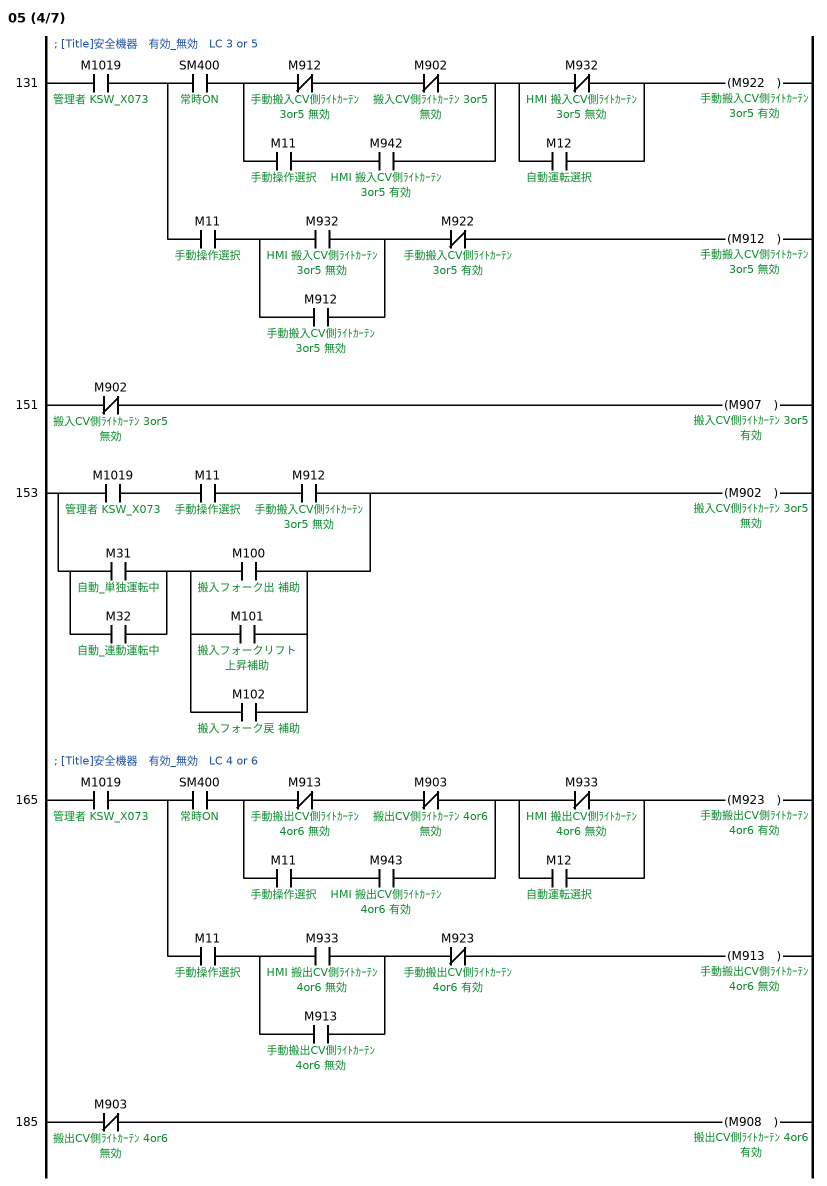
; [Title]安全機器　有効_無効　LC 3 or 5
131   LD      M1019  ; 管理者 KSW_X073
      MPS
      AND     SM400  ; 常時ON
      LDI     M912  ; 手動搬入CV側ﾗｲﾄｶｰﾃﾝ 3or5 無効
      ANI     M902  ; 搬入CV側ﾗｲﾄｶｰﾃﾝ 3or5 無効
      LD      M11  ; 手動操作選択
      AND     M942  ; HMI 搬入CV側ﾗｲﾄｶｰﾃﾝ 3or5 有効
      ORB
      ANB
      LDI     M932  ; HMI 搬入CV側ﾗｲﾄｶｰﾃﾝ 3or5 無効
      OR      M12  ; 自動運転選択
      ANB
      OUT     M922  ; 手動搬入CV側ﾗｲﾄｶｰﾃﾝ 3or5 有効
      MPP
      AND     M11  ; 手動操作選択
      LD      M932  ; HMI 搬入CV側ﾗｲﾄｶｰﾃﾝ 3or5 無効
      OR      M912  ; 手動搬入CV側ﾗｲﾄｶｰﾃﾝ 3or5 無効
      ANB
      ANI     M922  ; 手動搬入CV側ﾗｲﾄｶｰﾃﾝ 3or5 有効
      OUT     M912  ; 手動搬入CV側ﾗｲﾄｶｰﾃﾝ 3or5 無効
151   LDI     M902  ; 搬入CV側ﾗｲﾄｶｰﾃﾝ 3or5 無効
      OUT     M907  ; 搬入CV側ﾗｲﾄｶｰﾃﾝ 3or5 有効
153   LD      M1019  ; 管理者 KSW_X073
      AND     M11  ; 手動操作選択
      AND     M912  ; 手動搬入CV側ﾗｲﾄｶｰﾃﾝ 3or5 無効
      LD      M31  ; 自動_単独運転中
      OR      M32  ; 自動_連動運転中
      LD      M100  ; 搬入フォーク出 補助
      OR      M101  ; 搬入フォークリフト 上昇補助
      OR      M102  ; 搬入フォーク戻 補助
      ANB
      ORB
      OUT     M902  ; 搬入CV側ﾗｲﾄｶｰﾃﾝ 3or5 無効
; [Title]安全機器　有効_無効　LC 4 or 6
165   LD      M1019  ; 管理者 KSW_X073
      MPS
      AND     SM400  ; 常時ON
      LDI     M913  ; 手動搬出CV側ﾗｲﾄｶｰﾃﾝ 4or6 無効
      ANI     M903  ; 搬出CV側ﾗｲﾄｶｰﾃﾝ 4or6 無効
      LD      M11  ; 手動操作選択
      AND     M943  ; HMI 搬出CV側ﾗｲﾄｶｰﾃﾝ 4or6 有効
      ORB
      ANB
      LDI     M933  ; HMI 搬出CV側ﾗｲﾄｶｰﾃﾝ 4or6 無効
      OR      M12  ; 自動運転選択
      ANB
      OUT     M923  ; 手動搬出CV側ﾗｲﾄｶｰﾃﾝ 4or6 有効
      MPP
      AND     M11  ; 手動操作選択
      LD      M933  ; HMI 搬出CV側ﾗｲﾄｶｰﾃﾝ 4or6 無効
      OR      M913  ; 手動搬出CV側ﾗｲﾄｶｰﾃﾝ 4or6 無効
      ANB
      ANI     M923  ; 手動搬出CV側ﾗｲﾄｶｰﾃﾝ 4or6 有効
      OUT     M913  ; 手動搬出CV側ﾗｲﾄｶｰﾃﾝ 4or6 無効
185   LDI     M903  ; 搬出CV側ﾗｲﾄｶｰﾃﾝ 4or6 無効
      OUT     M908  ; 搬出CV側ﾗｲﾄｶｰﾃﾝ 4or6 有効
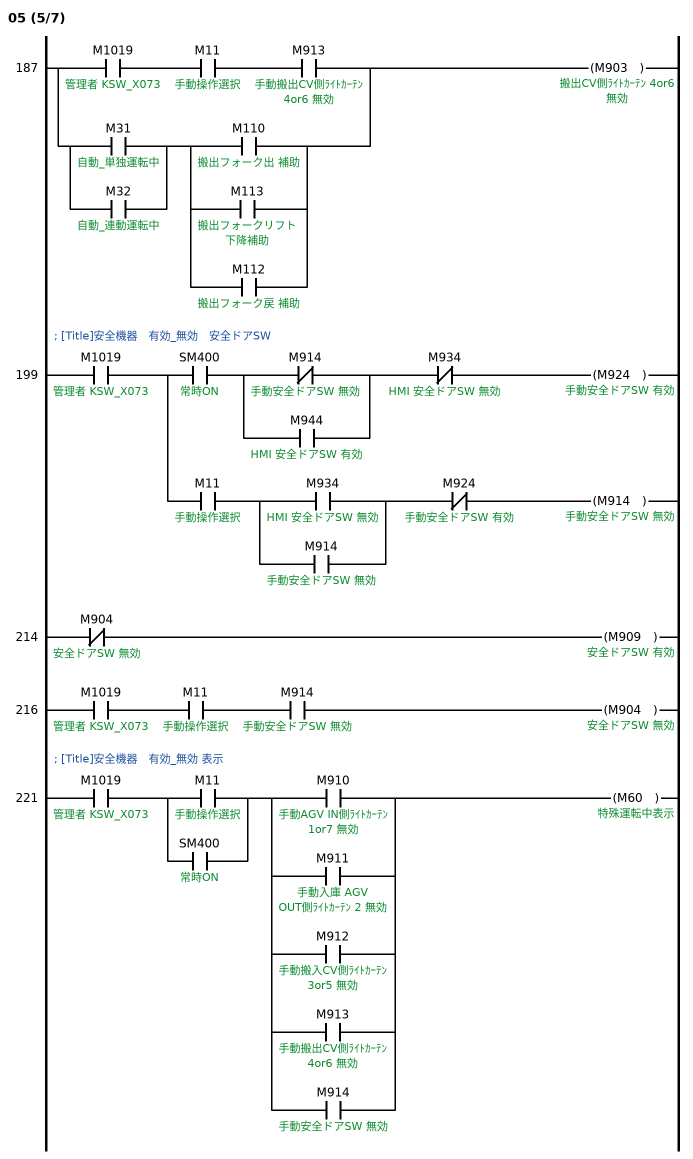
187   LD      M1019  ; 管理者 KSW_X073
      AND     M11  ; 手動操作選択
      AND     M913  ; 手動搬出CV側ﾗｲﾄｶｰﾃﾝ 4or6 無効
      LD      M31  ; 自動_単独運転中
      OR      M32  ; 自動_連動運転中
      LD      M110  ; 搬出フォーク出 補助
      OR      M113  ; 搬出フォークリフト 下降補助
      OR      M112  ; 搬出フォーク戻 補助
      ANB
      ORB
      OUT     M903  ; 搬出CV側ﾗｲﾄｶｰﾃﾝ 4or6 無効
; [Title]安全機器　有効_無効　安全ドアSW
199   LD      M1019  ; 管理者 KSW_X073
      MPS
      AND     SM400  ; 常時ON
      LDI     M914  ; 手動安全ドアSW 無効
      OR      M944  ; HMI 安全ドアSW 有効
      ANB
      ANI     M934  ; HMI 安全ドアSW 無効
      OUT     M924  ; 手動安全ドアSW 有効
      MPP
      AND     M11  ; 手動操作選択
      LD      M934  ; HMI 安全ドアSW 無効
      OR      M914  ; 手動安全ドアSW 無効
      ANB
      ANI     M924  ; 手動安全ドアSW 有効
      OUT     M914  ; 手動安全ドアSW 無効
214   LDI     M904  ; 安全ドアSW 無効
      OUT     M909  ; 安全ドアSW 有効
216   LD      M1019  ; 管理者 KSW_X073
      AND     M11  ; 手動操作選択
      AND     M914  ; 手動安全ドアSW 無効
      OUT     M904  ; 安全ドアSW 無効
; [Title]安全機器　有効_無効 表示
221   LD      M1019  ; 管理者 KSW_X073
      LD      M11  ; 手動操作選択
      OR      SM400  ; 常時ON
      ANB
      LD      M910  ; 手動AGV IN側ﾗｲﾄｶｰﾃﾝ 1or7 無効
      OR      M911  ; 手動入庫 AGV OUT側ﾗｲﾄｶｰﾃﾝ 2 無効
      OR      M912  ; 手動搬入CV側ﾗｲﾄｶｰﾃﾝ 3or5 無効
      OR      M913  ; 手動搬出CV側ﾗｲﾄｶｰﾃﾝ 4or6 無効
      OR      M914  ; 手動安全ドアSW 無効
      ANB
      OUT     M60  ; 特殊運転中表示
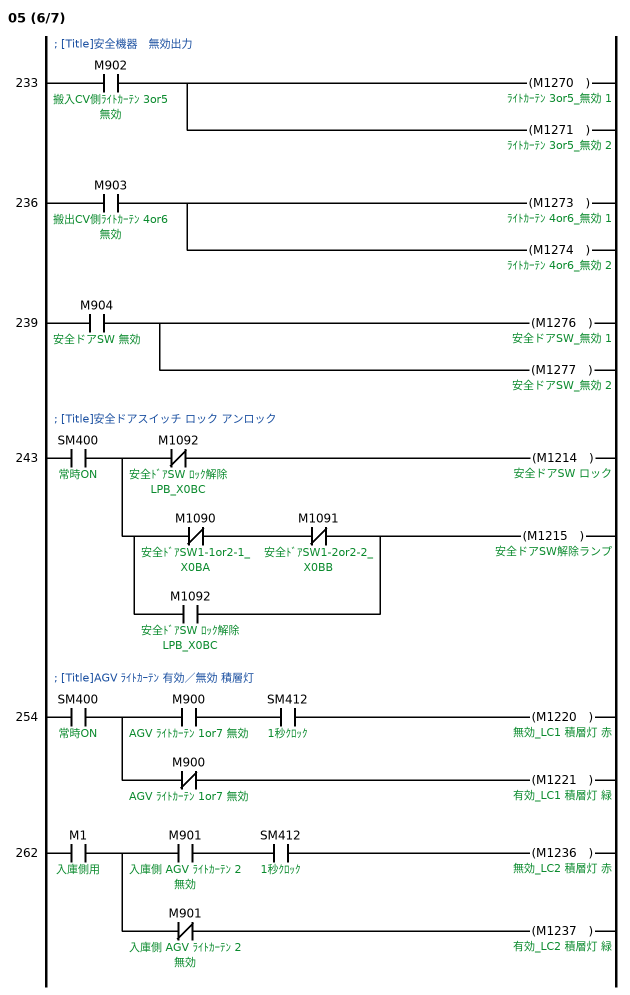
; [Title]安全機器　無効出力
233   LD      M902  ; 搬入CV側ﾗｲﾄｶｰﾃﾝ 3or5 無効
      OUT     M1270  ; ﾗｲﾄｶｰﾃﾝ 3or5_無効 1
      OUT     M1271  ; ﾗｲﾄｶｰﾃﾝ 3or5_無効 2
236   LD      M903  ; 搬出CV側ﾗｲﾄｶｰﾃﾝ 4or6 無効
      OUT     M1273  ; ﾗｲﾄｶｰﾃﾝ 4or6_無効 1
      OUT     M1274  ; ﾗｲﾄｶｰﾃﾝ 4or6_無効 2
239   LD      M904  ; 安全ドアSW 無効
      OUT     M1276  ; 安全ドアSW_無効 1
      OUT     M1277  ; 安全ドアSW_無効 2
; [Title]安全ドアスイッチ ロック アンロック
243   LD      SM400  ; 常時ON
      MPS
      ANI     M1092  ; 安全ﾄﾞｱSW ﾛｯｸ解除 LPB_X0BC
      OUT     M1214  ; 安全ドアSW ロック
      MPP
      LDI     M1090  ; 安全ﾄﾞｱSW1-1or2-1_X0BA
      ANI     M1091  ; 安全ﾄﾞｱSW1-2or2-2_X0BB
      OR      M1092  ; 安全ﾄﾞｱSW ﾛｯｸ解除 LPB_X0BC
      ANB
      OUT     M1215  ; 安全ドアSW解除ランプ
; [Title]AGV ﾗｲﾄｶｰﾃﾝ 有効／無効 積層灯
254   LD      SM400  ; 常時ON
      MPS
      AND     M900  ; AGV ﾗｲﾄｶｰﾃﾝ 1or7 無効
      AND     SM412  ; 1秒ｸﾛｯｸ
      OUT     M1220  ; 無効_LC1 積層灯 赤
      MPP
      ANI     M900  ; AGV ﾗｲﾄｶｰﾃﾝ 1or7 無効
      OUT     M1221  ; 有効_LC1 積層灯 緑
262   LD      M1  ; 入庫側用
      MPS
      AND     M901  ; 入庫側 AGV ﾗｲﾄｶｰﾃﾝ 2 無効
      AND     SM412  ; 1秒ｸﾛｯｸ
      OUT     M1236  ; 無効_LC2 積層灯 赤
      MPP
      ANI     M901  ; 入庫側 AGV ﾗｲﾄｶｰﾃﾝ 2 無効
      OUT     M1237  ; 有効_LC2 積層灯 緑
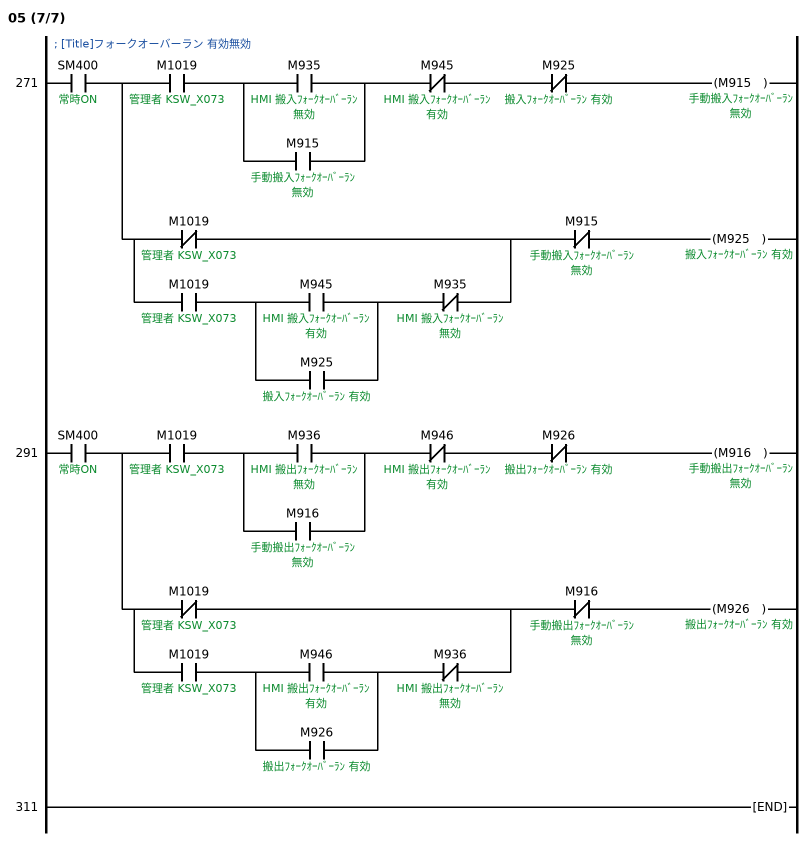
; [Title]フォークオーバーラン 有効無効
271   LD      SM400  ; 常時ON
      MPS
      AND     M1019  ; 管理者 KSW_X073
      LD      M935  ; HMI 搬入ﾌｫｰｸｵｰﾊﾞｰﾗﾝ 無効
      OR      M915  ; 手動搬入ﾌｫｰｸｵｰﾊﾞｰﾗﾝ 無効
      ANB
      ANI     M945  ; HMI 搬入ﾌｫｰｸｵｰﾊﾞｰﾗﾝ 有効
      ANI     M925  ; 搬入ﾌｫｰｸｵｰﾊﾞｰﾗﾝ 有効
      OUT     M915  ; 手動搬入ﾌｫｰｸｵｰﾊﾞｰﾗﾝ 無効
      MPP
      LDI     M1019  ; 管理者 KSW_X073
      LD      M1019  ; 管理者 KSW_X073
      LD      M945  ; HMI 搬入ﾌｫｰｸｵｰﾊﾞｰﾗﾝ 有効
      OR      M925  ; 搬入ﾌｫｰｸｵｰﾊﾞｰﾗﾝ 有効
      ANB
      ANI     M935  ; HMI 搬入ﾌｫｰｸｵｰﾊﾞｰﾗﾝ 無効
      ORB
      ANB
      ANI     M915  ; 手動搬入ﾌｫｰｸｵｰﾊﾞｰﾗﾝ 無効
      OUT     M925  ; 搬入ﾌｫｰｸｵｰﾊﾞｰﾗﾝ 有効
291   LD      SM400  ; 常時ON
      MPS
      AND     M1019  ; 管理者 KSW_X073
      LD      M936  ; HMI 搬出ﾌｫｰｸｵｰﾊﾞｰﾗﾝ 無効
      OR      M916  ; 手動搬出ﾌｫｰｸｵｰﾊﾞｰﾗﾝ 無効
      ANB
      ANI     M946  ; HMI 搬出ﾌｫｰｸｵｰﾊﾞｰﾗﾝ 有効
      ANI     M926  ; 搬出ﾌｫｰｸｵｰﾊﾞｰﾗﾝ 有効
      OUT     M916  ; 手動搬出ﾌｫｰｸｵｰﾊﾞｰﾗﾝ 無効
      MPP
      LDI     M1019  ; 管理者 KSW_X073
      LD      M1019  ; 管理者 KSW_X073
      LD      M946  ; HMI 搬出ﾌｫｰｸｵｰﾊﾞｰﾗﾝ 有効
      OR      M926  ; 搬出ﾌｫｰｸｵｰﾊﾞｰﾗﾝ 有効
      ANB
      ANI     M936  ; HMI 搬出ﾌｫｰｸｵｰﾊﾞｰﾗﾝ 無効
      ORB
      ANB
      ANI     M916  ; 手動搬出ﾌｫｰｸｵｰﾊﾞｰﾗﾝ 無効
      OUT     M926  ; 搬出ﾌｫｰｸｵｰﾊﾞｰﾗﾝ 有効
311   END
END_PROGRAM

PROGRAM 09  // Alram
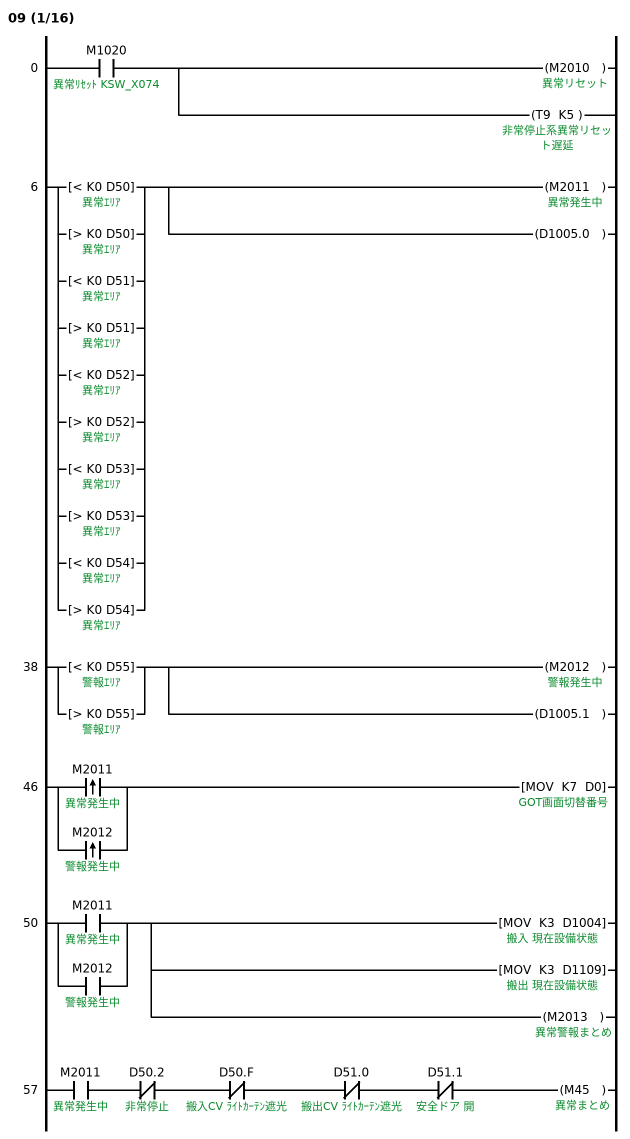
0     LD      M1020  ; 異常ﾘｾｯﾄ KSW_X074
      OUT     M2010  ; 異常リセット
      OUT     T9 K5  ; 非常停止系異常リセット遅延
6     LD<     K0 D50  ; 異常ｴﾘｱ
      OR>     K0 D50  ; 異常ｴﾘｱ
      OR<     K0 D51  ; 異常ｴﾘｱ
      OR>     K0 D51  ; 異常ｴﾘｱ
      OR<     K0 D52  ; 異常ｴﾘｱ
      OR>     K0 D52  ; 異常ｴﾘｱ
      OR<     K0 D53  ; 異常ｴﾘｱ
      OR>     K0 D53  ; 異常ｴﾘｱ
      OR<     K0 D54  ; 異常ｴﾘｱ
      OR>     K0 D54  ; 異常ｴﾘｱ
      OUT     M2011  ; 異常発生中
      OUT     D1005.0
38    LD<     K0 D55  ; 警報ｴﾘｱ
      OR>     K0 D55  ; 警報ｴﾘｱ
      OUT     M2012  ; 警報発生中
      OUT     D1005.1
46    LDP     M2011  ; 異常発生中
      ORP     M2012  ; 警報発生中
      MOV     K7 D0  ; GOT画面切替番号
50    LD      M2011  ; 異常発生中
      OR      M2012  ; 警報発生中
      MOV     K3 D1004  ; 搬入 現在設備状態
      MOV     K3 D1109  ; 搬出 現在設備状態
      OUT     M2013  ; 異常警報まとめ
57    LD      M2011  ; 異常発生中
      ANI     D50.2  ; 非常停止
      ANI     D50.F  ; 搬入CV ﾗｲﾄｶｰﾃﾝ遮光
      ANI     D51.0  ; 搬出CV ﾗｲﾄｶｰﾃﾝ遮光
      ANI     D51.1  ; 安全ドア 開
      OUT     M45  ; 異常まとめ
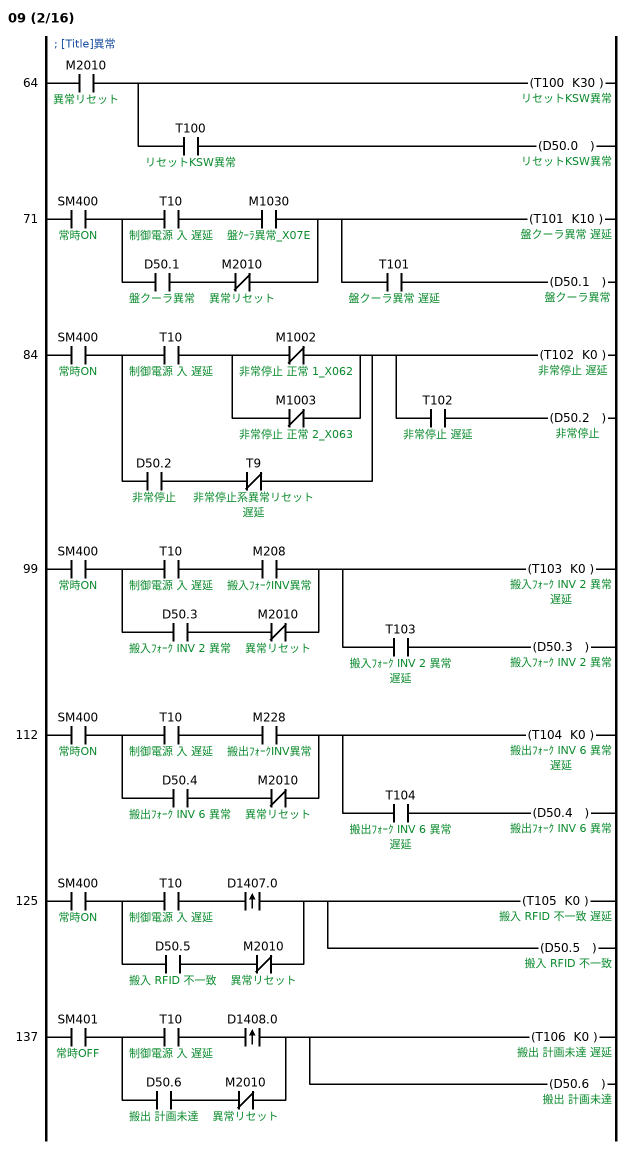
; [Title]異常
64    LD      M2010  ; 異常リセット
      OUT     T100 K30  ; リセットKSW異常
      AND     T100  ; リセットKSW異常
      OUT     D50.0  ; リセットKSW異常
71    LD      SM400  ; 常時ON
      LD      T10  ; 制御電源 入 遅延
      AND     M1030  ; 盤ｸｰﾗ異常_X07E
      LD      D50.1  ; 盤クーラ異常
      ANI     M2010  ; 異常リセット
      ORB
      ANB
      OUT     T101 K10  ; 盤クーラ異常 遅延
      AND     T101  ; 盤クーラ異常 遅延
      OUT     D50.1  ; 盤クーラ異常
84    LD      SM400  ; 常時ON
      LD      T10  ; 制御電源 入 遅延
      LDI     M1002  ; 非常停止 正常 1_X062
      ORI     M1003  ; 非常停止 正常 2_X063
      ANB
      LD      D50.2  ; 非常停止
      ANI     T9  ; 非常停止系異常リセット遅延
      ORB
      ANB
      OUT     T102 K0  ; 非常停止 遅延
      AND     T102  ; 非常停止 遅延
      OUT     D50.2  ; 非常停止
99    LD      SM400  ; 常時ON
      LD      T10  ; 制御電源 入 遅延
      AND     M208  ; 搬入ﾌｫｰｸINV異常
      LD      D50.3  ; 搬入ﾌｫｰｸ INV 2 異常
      ANI     M2010  ; 異常リセット
      ORB
      ANB
      OUT     T103 K0  ; 搬入ﾌｫｰｸ INV 2 異常 遅延
      AND     T103  ; 搬入ﾌｫｰｸ INV 2 異常 遅延
      OUT     D50.3  ; 搬入ﾌｫｰｸ INV 2 異常
112   LD      SM400  ; 常時ON
      LD      T10  ; 制御電源 入 遅延
      AND     M228  ; 搬出ﾌｫｰｸINV異常
      LD      D50.4  ; 搬出ﾌｫｰｸ INV 6 異常
      ANI     M2010  ; 異常リセット
      ORB
      ANB
      OUT     T104 K0  ; 搬出ﾌｫｰｸ INV 6 異常 遅延
      AND     T104  ; 搬出ﾌｫｰｸ INV 6 異常 遅延
      OUT     D50.4  ; 搬出ﾌｫｰｸ INV 6 異常
125   LD      SM400  ; 常時ON
      LD      T10  ; 制御電源 入 遅延
      ANDP    D1407.0
      LD      D50.5  ; 搬入 RFID 不一致
      ANI     M2010  ; 異常リセット
      ORB
      ANB
      OUT     T105 K0  ; 搬入 RFID 不一致 遅延
      OUT     D50.5  ; 搬入 RFID 不一致
137   LD      SM401  ; 常時OFF
      LD      T10  ; 制御電源 入 遅延
      ANDP    D1408.0
      LD      D50.6  ; 搬出 計画未達
      ANI     M2010  ; 異常リセット
      ORB
      ANB
      OUT     T106 K0  ; 搬出 計画未達 遅延
      OUT     D50.6  ; 搬出 計画未達
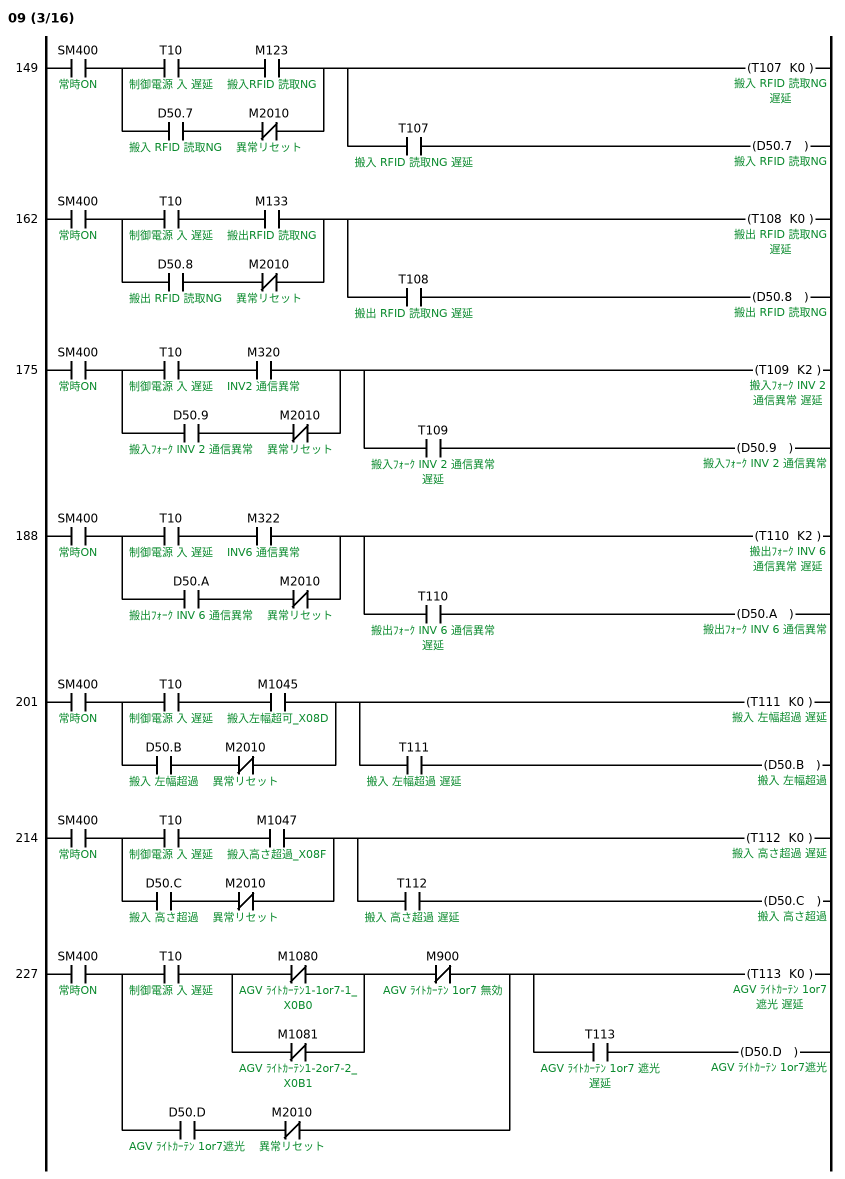
149   LD      SM400  ; 常時ON
      LD      T10  ; 制御電源 入 遅延
      AND     M123  ; 搬入RFID 読取NG
      LD      D50.7  ; 搬入 RFID 読取NG
      ANI     M2010  ; 異常リセット
      ORB
      ANB
      OUT     T107 K0  ; 搬入 RFID 読取NG 遅延
      AND     T107  ; 搬入 RFID 読取NG 遅延
      OUT     D50.7  ; 搬入 RFID 読取NG
162   LD      SM400  ; 常時ON
      LD      T10  ; 制御電源 入 遅延
      AND     M133  ; 搬出RFID 読取NG
      LD      D50.8  ; 搬出 RFID 読取NG
      ANI     M2010  ; 異常リセット
      ORB
      ANB
      OUT     T108 K0  ; 搬出 RFID 読取NG 遅延
      AND     T108  ; 搬出 RFID 読取NG 遅延
      OUT     D50.8  ; 搬出 RFID 読取NG
175   LD      SM400  ; 常時ON
      LD      T10  ; 制御電源 入 遅延
      AND     M320  ; INV2 通信異常
      LD      D50.9  ; 搬入ﾌｫｰｸ INV 2 通信異常
      ANI     M2010  ; 異常リセット
      ORB
      ANB
      OUT     T109 K2  ; 搬入ﾌｫｰｸ INV 2 通信異常 遅延
      AND     T109  ; 搬入ﾌｫｰｸ INV 2 通信異常 遅延
      OUT     D50.9  ; 搬入ﾌｫｰｸ INV 2 通信異常
188   LD      SM400  ; 常時ON
      LD      T10  ; 制御電源 入 遅延
      AND     M322  ; INV6 通信異常
      LD      D50.A  ; 搬出ﾌｫｰｸ INV 6 通信異常
      ANI     M2010  ; 異常リセット
      ORB
      ANB
      OUT     T110 K2  ; 搬出ﾌｫｰｸ INV 6 通信異常 遅延
      AND     T110  ; 搬出ﾌｫｰｸ INV 6 通信異常 遅延
      OUT     D50.A  ; 搬出ﾌｫｰｸ INV 6 通信異常
201   LD      SM400  ; 常時ON
      LD      T10  ; 制御電源 入 遅延
      AND     M1045  ; 搬入左幅超可_X08D
      LD      D50.B  ; 搬入 左幅超過
      ANI     M2010  ; 異常リセット
      ORB
      ANB
      OUT     T111 K0  ; 搬入 左幅超過 遅延
      AND     T111  ; 搬入 左幅超過 遅延
      OUT     D50.B  ; 搬入 左幅超過
214   LD      SM400  ; 常時ON
      LD      T10  ; 制御電源 入 遅延
      AND     M1047  ; 搬入高さ超過_X08F
      LD      D50.C  ; 搬入 高さ超過
      ANI     M2010  ; 異常リセット
      ORB
      ANB
      OUT     T112 K0  ; 搬入 高さ超過 遅延
      AND     T112  ; 搬入 高さ超過 遅延
      OUT     D50.C  ; 搬入 高さ超過
227   LD      SM400  ; 常時ON
      LD      T10  ; 制御電源 入 遅延
      LDI     M1080  ; AGV ﾗｲﾄｶｰﾃﾝ1-1or7-1_X0B0
      ORI     M1081  ; AGV ﾗｲﾄｶｰﾃﾝ1-2or7-2_X0B1
      ANB
      ANI     M900  ; AGV ﾗｲﾄｶｰﾃﾝ 1or7 無効
      LD      D50.D  ; AGV ﾗｲﾄｶｰﾃﾝ 1or7遮光
      ANI     M2010  ; 異常リセット
      ORB
      ANB
      OUT     T113 K0  ; AGV ﾗｲﾄｶｰﾃﾝ 1or7 遮光 遅延
      AND     T113  ; AGV ﾗｲﾄｶｰﾃﾝ 1or7 遮光 遅延
      OUT     D50.D  ; AGV ﾗｲﾄｶｰﾃﾝ 1or7遮光
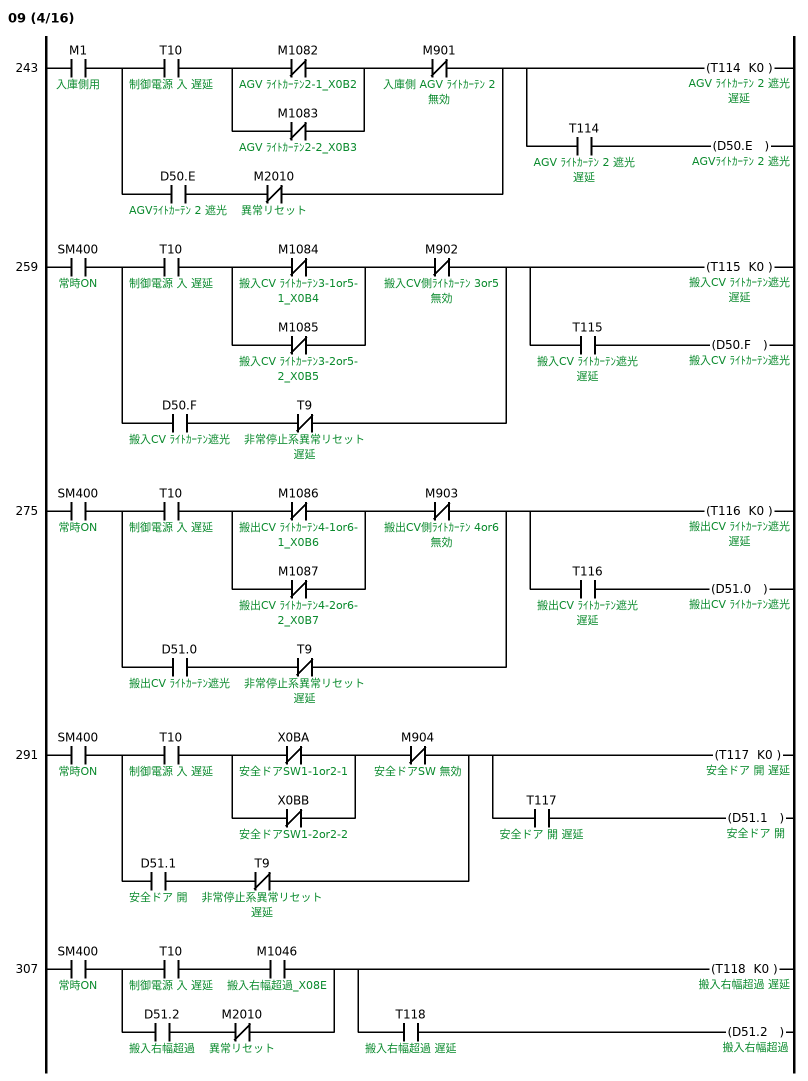
243   LD      M1  ; 入庫側用
      LD      T10  ; 制御電源 入 遅延
      LDI     M1082  ; AGV ﾗｲﾄｶｰﾃﾝ2-1_X0B2
      ORI     M1083  ; AGV ﾗｲﾄｶｰﾃﾝ2-2_X0B3
      ANB
      ANI     M901  ; 入庫側 AGV ﾗｲﾄｶｰﾃﾝ 2 無効
      LD      D50.E  ; AGVﾗｲﾄｶｰﾃﾝ 2 遮光
      ANI     M2010  ; 異常リセット
      ORB
      ANB
      OUT     T114 K0  ; AGV ﾗｲﾄｶｰﾃﾝ 2 遮光 遅延
      AND     T114  ; AGV ﾗｲﾄｶｰﾃﾝ 2 遮光 遅延
      OUT     D50.E  ; AGVﾗｲﾄｶｰﾃﾝ 2 遮光
259   LD      SM400  ; 常時ON
      LD      T10  ; 制御電源 入 遅延
      LDI     M1084  ; 搬入CV ﾗｲﾄｶｰﾃﾝ3-1or5-1_X0B4
      ORI     M1085  ; 搬入CV ﾗｲﾄｶｰﾃﾝ3-2or5-2_X0B5
      ANB
      ANI     M902  ; 搬入CV側ﾗｲﾄｶｰﾃﾝ 3or5 無効
      LD      D50.F  ; 搬入CV ﾗｲﾄｶｰﾃﾝ遮光
      ANI     T9  ; 非常停止系異常リセット遅延
      ORB
      ANB
      OUT     T115 K0  ; 搬入CV ﾗｲﾄｶｰﾃﾝ遮光 遅延
      AND     T115  ; 搬入CV ﾗｲﾄｶｰﾃﾝ遮光 遅延
      OUT     D50.F  ; 搬入CV ﾗｲﾄｶｰﾃﾝ遮光
275   LD      SM400  ; 常時ON
      LD      T10  ; 制御電源 入 遅延
      LDI     M1086  ; 搬出CV ﾗｲﾄｶｰﾃﾝ4-1or6-1_X0B6
      ORI     M1087  ; 搬出CV ﾗｲﾄｶｰﾃﾝ4-2or6-2_X0B7
      ANB
      ANI     M903  ; 搬出CV側ﾗｲﾄｶｰﾃﾝ 4or6 無効
      LD      D51.0  ; 搬出CV ﾗｲﾄｶｰﾃﾝ遮光
      ANI     T9  ; 非常停止系異常リセット遅延
      ORB
      ANB
      OUT     T116 K0  ; 搬出CV ﾗｲﾄｶｰﾃﾝ遮光 遅延
      AND     T116  ; 搬出CV ﾗｲﾄｶｰﾃﾝ遮光 遅延
      OUT     D51.0  ; 搬出CV ﾗｲﾄｶｰﾃﾝ遮光
291   LD      SM400  ; 常時ON
      LD      T10  ; 制御電源 入 遅延
      LDI     X0BA  ; 安全ドアSW1-1or2-1
      ORI     X0BB  ; 安全ドアSW1-2or2-2
      ANB
      ANI     M904  ; 安全ドアSW 無効
      LD      D51.1  ; 安全ドア 開
      ANI     T9  ; 非常停止系異常リセット遅延
      ORB
      ANB
      OUT     T117 K0  ; 安全ドア 開 遅延
      AND     T117  ; 安全ドア 開 遅延
      OUT     D51.1  ; 安全ドア 開
307   LD      SM400  ; 常時ON
      LD      T10  ; 制御電源 入 遅延
      AND     M1046  ; 搬入右幅超過_X08E
      LD      D51.2  ; 搬入右幅超過
      ANI     M2010  ; 異常リセット
      ORB
      ANB
      OUT     T118 K0  ; 搬入右幅超過 遅延
      AND     T118  ; 搬入右幅超過 遅延
      OUT     D51.2  ; 搬入右幅超過
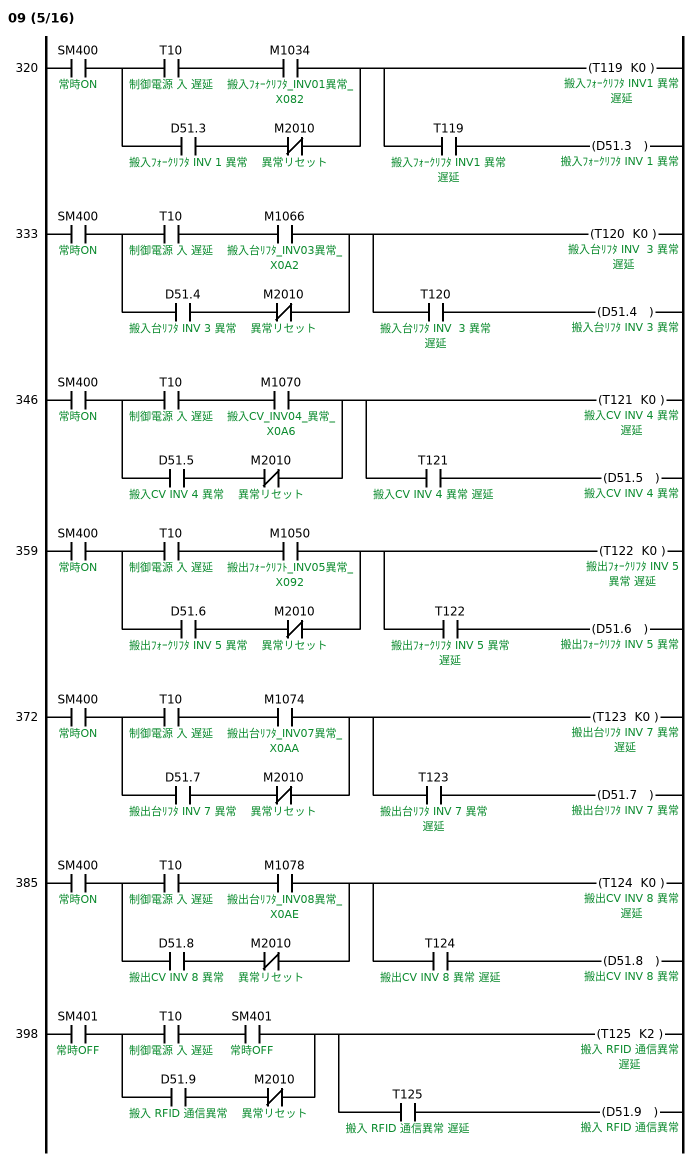
320   LD      SM400  ; 常時ON
      LD      T10  ; 制御電源 入 遅延
      AND     M1034  ; 搬入ﾌｫｰｸﾘﾌﾀ_INV01異常_X082
      LD      D51.3  ; 搬入ﾌｫｰｸﾘﾌﾀ INV 1 異常
      ANI     M2010  ; 異常リセット
      ORB
      ANB
      OUT     T119 K0  ; 搬入ﾌｫｰｸﾘﾌﾀ INV1 異常 遅延
      AND     T119  ; 搬入ﾌｫｰｸﾘﾌﾀ INV1 異常 遅延
      OUT     D51.3  ; 搬入ﾌｫｰｸﾘﾌﾀ INV 1 異常
333   LD      SM400  ; 常時ON
      LD      T10  ; 制御電源 入 遅延
      AND     M1066  ; 搬入台ﾘﾌﾀ_INV03異常_X0A2
      LD      D51.4  ; 搬入台ﾘﾌﾀ INV 3 異常
      ANI     M2010  ; 異常リセット
      ORB
      ANB
      OUT     T120 K0  ; 搬入台ﾘﾌﾀ INV  3 異常 遅延
      AND     T120  ; 搬入台ﾘﾌﾀ INV  3 異常 遅延
      OUT     D51.4  ; 搬入台ﾘﾌﾀ INV 3 異常
346   LD      SM400  ; 常時ON
      LD      T10  ; 制御電源 入 遅延
      AND     M1070  ; 搬入CV_INV04_異常_X0A6
      LD      D51.5  ; 搬入CV INV 4 異常
      ANI     M2010  ; 異常リセット
      ORB
      ANB
      OUT     T121 K0  ; 搬入CV INV 4 異常 遅延
      AND     T121  ; 搬入CV INV 4 異常 遅延
      OUT     D51.5  ; 搬入CV INV 4 異常
359   LD      SM400  ; 常時ON
      LD      T10  ; 制御電源 入 遅延
      AND     M1050  ; 搬出ﾌｫｰｸﾘﾌﾄ_INV05異常_X092
      LD      D51.6  ; 搬出ﾌｫｰｸﾘﾌﾀ INV 5 異常
      ANI     M2010  ; 異常リセット
      ORB
      ANB
      OUT     T122 K0  ; 搬出ﾌｫｰｸﾘﾌﾀ INV 5 異常 遅延
      AND     T122  ; 搬出ﾌｫｰｸﾘﾌﾀ INV 5 異常 遅延
      OUT     D51.6  ; 搬出ﾌｫｰｸﾘﾌﾀ INV 5 異常
372   LD      SM400  ; 常時ON
      LD      T10  ; 制御電源 入 遅延
      AND     M1074  ; 搬出台ﾘﾌﾀ_INV07異常_X0AA
      LD      D51.7  ; 搬出台ﾘﾌﾀ INV 7 異常
      ANI     M2010  ; 異常リセット
      ORB
      ANB
      OUT     T123 K0  ; 搬出台ﾘﾌﾀ INV 7 異常 遅延
      AND     T123  ; 搬出台ﾘﾌﾀ INV 7 異常 遅延
      OUT     D51.7  ; 搬出台ﾘﾌﾀ INV 7 異常
385   LD      SM400  ; 常時ON
      LD      T10  ; 制御電源 入 遅延
      AND     M1078  ; 搬出台ﾘﾌﾀ_INV08異常_X0AE
      LD      D51.8  ; 搬出CV INV 8 異常
      ANI     M2010  ; 異常リセット
      ORB
      ANB
      OUT     T124 K0  ; 搬出CV INV 8 異常 遅延
      AND     T124  ; 搬出CV INV 8 異常 遅延
      OUT     D51.8  ; 搬出CV INV 8 異常
398   LD      SM401  ; 常時OFF
      LD      T10  ; 制御電源 入 遅延
      AND     SM401  ; 常時OFF
      LD      D51.9  ; 搬入 RFID 通信異常
      ANI     M2010  ; 異常リセット
      ORB
      ANB
      OUT     T125 K2  ; 搬入 RFID 通信異常 遅延
      AND     T125  ; 搬入 RFID 通信異常 遅延
      OUT     D51.9  ; 搬入 RFID 通信異常
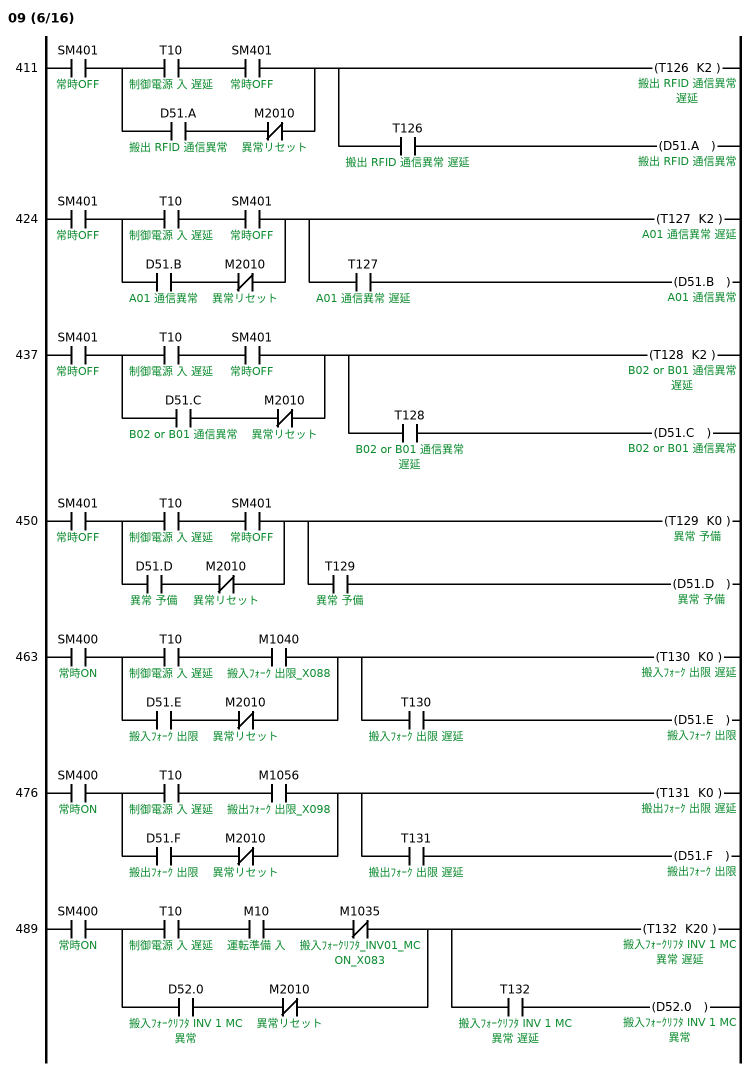
411   LD      SM401  ; 常時OFF
      LD      T10  ; 制御電源 入 遅延
      AND     SM401  ; 常時OFF
      LD      D51.A  ; 搬出 RFID 通信異常
      ANI     M2010  ; 異常リセット
      ORB
      ANB
      OUT     T126 K2  ; 搬出 RFID 通信異常 遅延
      AND     T126  ; 搬出 RFID 通信異常 遅延
      OUT     D51.A  ; 搬出 RFID 通信異常
424   LD      SM401  ; 常時OFF
      LD      T10  ; 制御電源 入 遅延
      AND     SM401  ; 常時OFF
      LD      D51.B  ; A01 通信異常
      ANI     M2010  ; 異常リセット
      ORB
      ANB
      OUT     T127 K2  ; A01 通信異常 遅延
      AND     T127  ; A01 通信異常 遅延
      OUT     D51.B  ; A01 通信異常
437   LD      SM401  ; 常時OFF
      LD      T10  ; 制御電源 入 遅延
      AND     SM401  ; 常時OFF
      LD      D51.C  ; B02 or B01 通信異常
      ANI     M2010  ; 異常リセット
      ORB
      ANB
      OUT     T128 K2  ; B02 or B01 通信異常 遅延
      AND     T128  ; B02 or B01 通信異常 遅延
      OUT     D51.C  ; B02 or B01 通信異常
450   LD      SM401  ; 常時OFF
      LD      T10  ; 制御電源 入 遅延
      AND     SM401  ; 常時OFF
      LD      D51.D  ; 異常 予備
      ANI     M2010  ; 異常リセット
      ORB
      ANB
      OUT     T129 K0  ; 異常 予備
      AND     T129  ; 異常 予備
      OUT     D51.D  ; 異常 予備
463   LD      SM400  ; 常時ON
      LD      T10  ; 制御電源 入 遅延
      AND     M1040  ; 搬入ﾌｫｰｸ 出限_X088
      LD      D51.E  ; 搬入ﾌｫｰｸ 出限
      ANI     M2010  ; 異常リセット
      ORB
      ANB
      OUT     T130 K0  ; 搬入ﾌｫｰｸ 出限 遅延
      AND     T130  ; 搬入ﾌｫｰｸ 出限 遅延
      OUT     D51.E  ; 搬入ﾌｫｰｸ 出限
476   LD      SM400  ; 常時ON
      LD      T10  ; 制御電源 入 遅延
      AND     M1056  ; 搬出ﾌｫｰｸ 出限_X098
      LD      D51.F  ; 搬出ﾌｫｰｸ 出限
      ANI     M2010  ; 異常リセット
      ORB
      ANB
      OUT     T131 K0  ; 搬出ﾌｫｰｸ 出限 遅延
      AND     T131  ; 搬出ﾌｫｰｸ 出限 遅延
      OUT     D51.F  ; 搬出ﾌｫｰｸ 出限
489   LD      SM400  ; 常時ON
      LD      T10  ; 制御電源 入 遅延
      AND     M10  ; 運転準備 入
      ANI     M1035  ; 搬入ﾌｫｰｸﾘﾌﾀ_INV01_MC ON_X083
      LD      D52.0  ; 搬入ﾌｫｰｸﾘﾌﾀ INV 1 MC 異常
      ANI     M2010  ; 異常リセット
      ORB
      ANB
      OUT     T132 K20  ; 搬入ﾌｫｰｸﾘﾌﾀ INV 1 MC 異常 遅延
      AND     T132  ; 搬入ﾌｫｰｸﾘﾌﾀ INV 1 MC 異常 遅延
      OUT     D52.0  ; 搬入ﾌｫｰｸﾘﾌﾀ INV 1 MC 異常
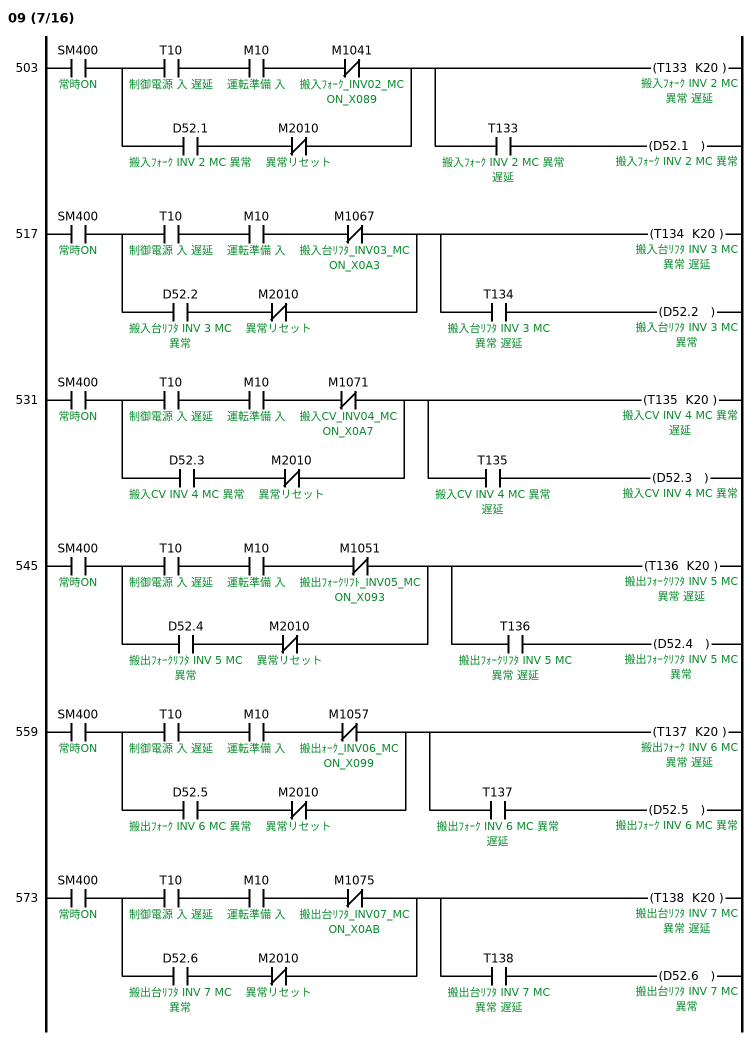
503   LD      SM400  ; 常時ON
      LD      T10  ; 制御電源 入 遅延
      AND     M10  ; 運転準備 入
      ANI     M1041  ; 搬入ﾌｫｰｸ_INV02_MC ON_X089
      LD      D52.1  ; 搬入ﾌｫｰｸ INV 2 MC 異常
      ANI     M2010  ; 異常リセット
      ORB
      ANB
      OUT     T133 K20  ; 搬入ﾌｫｰｸ INV 2 MC 異常 遅延
      AND     T133  ; 搬入ﾌｫｰｸ INV 2 MC 異常 遅延
      OUT     D52.1  ; 搬入ﾌｫｰｸ INV 2 MC 異常
517   LD      SM400  ; 常時ON
      LD      T10  ; 制御電源 入 遅延
      AND     M10  ; 運転準備 入
      ANI     M1067  ; 搬入台ﾘﾌﾀ_INV03_MC ON_X0A3
      LD      D52.2  ; 搬入台ﾘﾌﾀ INV 3 MC 異常
      ANI     M2010  ; 異常リセット
      ORB
      ANB
      OUT     T134 K20  ; 搬入台ﾘﾌﾀ INV 3 MC 異常 遅延
      AND     T134  ; 搬入台ﾘﾌﾀ INV 3 MC 異常 遅延
      OUT     D52.2  ; 搬入台ﾘﾌﾀ INV 3 MC 異常
531   LD      SM400  ; 常時ON
      LD      T10  ; 制御電源 入 遅延
      AND     M10  ; 運転準備 入
      ANI     M1071  ; 搬入CV_INV04_MC ON_X0A7
      LD      D52.3  ; 搬入CV INV 4 MC 異常
      ANI     M2010  ; 異常リセット
      ORB
      ANB
      OUT     T135 K20  ; 搬入CV INV 4 MC 異常 遅延
      AND     T135  ; 搬入CV INV 4 MC 異常 遅延
      OUT     D52.3  ; 搬入CV INV 4 MC 異常
545   LD      SM400  ; 常時ON
      LD      T10  ; 制御電源 入 遅延
      AND     M10  ; 運転準備 入
      ANI     M1051  ; 搬出ﾌｫｰｸﾘﾌﾄ_INV05_MC ON_X093
      LD      D52.4  ; 搬出ﾌｫｰｸﾘﾌﾀ INV 5 MC 異常
      ANI     M2010  ; 異常リセット
      ORB
      ANB
      OUT     T136 K20  ; 搬出ﾌｫｰｸﾘﾌﾀ INV 5 MC 異常 遅延
      AND     T136  ; 搬出ﾌｫｰｸﾘﾌﾀ INV 5 MC 異常 遅延
      OUT     D52.4  ; 搬出ﾌｫｰｸﾘﾌﾀ INV 5 MC 異常
559   LD      SM400  ; 常時ON
      LD      T10  ; 制御電源 入 遅延
      AND     M10  ; 運転準備 入
      ANI     M1057  ; 搬出ｫｰｸ_INV06_MC ON_X099
      LD      D52.5  ; 搬出ﾌｫｰｸ INV 6 MC 異常
      ANI     M2010  ; 異常リセット
      ORB
      ANB
      OUT     T137 K20  ; 搬出ﾌｫｰｸ INV 6 MC 異常 遅延
      AND     T137  ; 搬出ﾌｫｰｸ INV 6 MC 異常 遅延
      OUT     D52.5  ; 搬出ﾌｫｰｸ INV 6 MC 異常
573   LD      SM400  ; 常時ON
      LD      T10  ; 制御電源 入 遅延
      AND     M10  ; 運転準備 入
      ANI     M1075  ; 搬出台ﾘﾌﾀ_INV07_MC ON_X0AB
      LD      D52.6  ; 搬出台ﾘﾌﾀ INV 7 MC 異常
      ANI     M2010  ; 異常リセット
      ORB
      ANB
      OUT     T138 K20  ; 搬出台ﾘﾌﾀ INV 7 MC 異常 遅延
      AND     T138  ; 搬出台ﾘﾌﾀ INV 7 MC 異常 遅延
      OUT     D52.6  ; 搬出台ﾘﾌﾀ INV 7 MC 異常
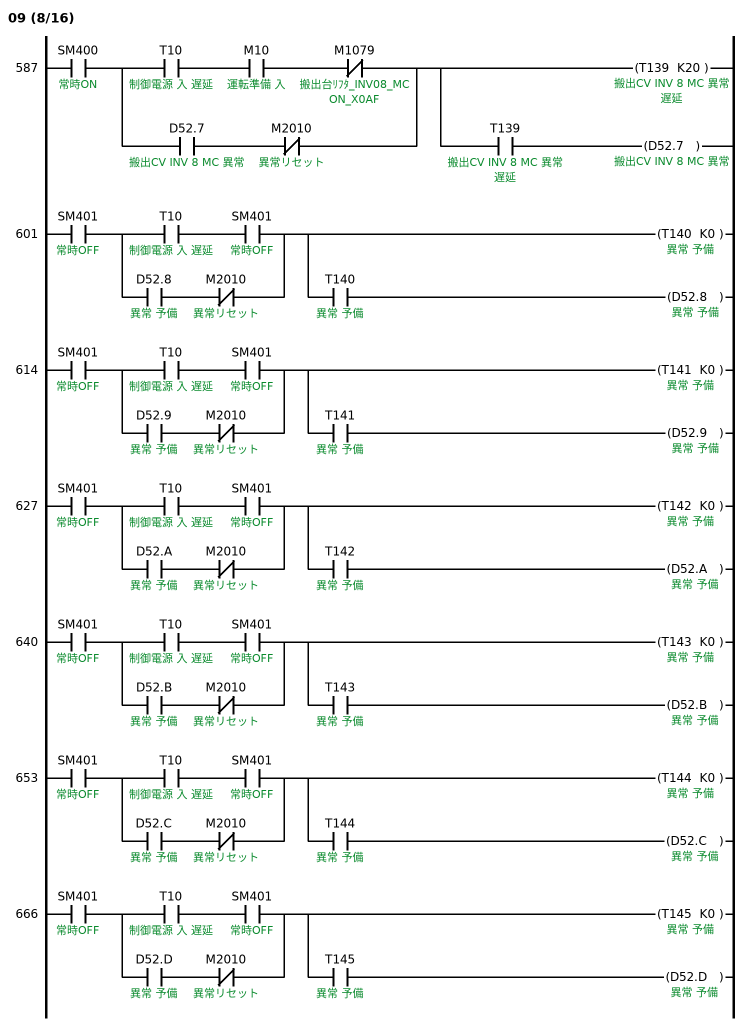
587   LD      SM400  ; 常時ON
      LD      T10  ; 制御電源 入 遅延
      AND     M10  ; 運転準備 入
      ANI     M1079  ; 搬出台ﾘﾌﾀ_INV08_MC ON_X0AF
      LD      D52.7  ; 搬出CV INV 8 MC 異常
      ANI     M2010  ; 異常リセット
      ORB
      ANB
      OUT     T139 K20  ; 搬出CV INV 8 MC 異常 遅延
      AND     T139  ; 搬出CV INV 8 MC 異常 遅延
      OUT     D52.7  ; 搬出CV INV 8 MC 異常
601   LD      SM401  ; 常時OFF
      LD      T10  ; 制御電源 入 遅延
      AND     SM401  ; 常時OFF
      LD      D52.8  ; 異常 予備
      ANI     M2010  ; 異常リセット
      ORB
      ANB
      OUT     T140 K0  ; 異常 予備
      AND     T140  ; 異常 予備
      OUT     D52.8  ; 異常 予備
614   LD      SM401  ; 常時OFF
      LD      T10  ; 制御電源 入 遅延
      AND     SM401  ; 常時OFF
      LD      D52.9  ; 異常 予備
      ANI     M2010  ; 異常リセット
      ORB
      ANB
      OUT     T141 K0  ; 異常 予備
      AND     T141  ; 異常 予備
      OUT     D52.9  ; 異常 予備
627   LD      SM401  ; 常時OFF
      LD      T10  ; 制御電源 入 遅延
      AND     SM401  ; 常時OFF
      LD      D52.A  ; 異常 予備
      ANI     M2010  ; 異常リセット
      ORB
      ANB
      OUT     T142 K0  ; 異常 予備
      AND     T142  ; 異常 予備
      OUT     D52.A  ; 異常 予備
640   LD      SM401  ; 常時OFF
      LD      T10  ; 制御電源 入 遅延
      AND     SM401  ; 常時OFF
      LD      D52.B  ; 異常 予備
      ANI     M2010  ; 異常リセット
      ORB
      ANB
      OUT     T143 K0  ; 異常 予備
      AND     T143  ; 異常 予備
      OUT     D52.B  ; 異常 予備
653   LD      SM401  ; 常時OFF
      LD      T10  ; 制御電源 入 遅延
      AND     SM401  ; 常時OFF
      LD      D52.C  ; 異常 予備
      ANI     M2010  ; 異常リセット
      ORB
      ANB
      OUT     T144 K0  ; 異常 予備
      AND     T144  ; 異常 予備
      OUT     D52.C  ; 異常 予備
666   LD      SM401  ; 常時OFF
      LD      T10  ; 制御電源 入 遅延
      AND     SM401  ; 常時OFF
      LD      D52.D  ; 異常 予備
      ANI     M2010  ; 異常リセット
      ORB
      ANB
      OUT     T145 K0  ; 異常 予備
      AND     T145  ; 異常 予備
      OUT     D52.D  ; 異常 予備
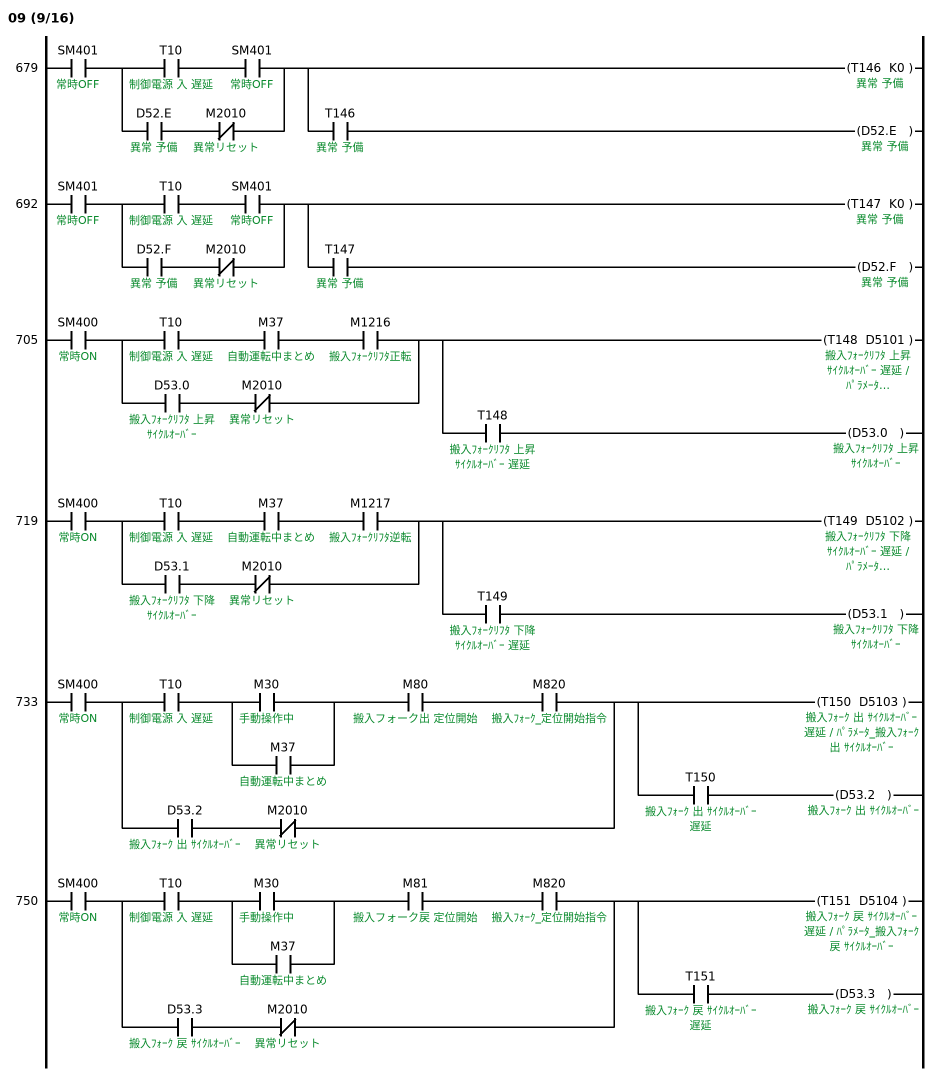
679   LD      SM401  ; 常時OFF
      LD      T10  ; 制御電源 入 遅延
      AND     SM401  ; 常時OFF
      LD      D52.E  ; 異常 予備
      ANI     M2010  ; 異常リセット
      ORB
      ANB
      OUT     T146 K0  ; 異常 予備
      AND     T146  ; 異常 予備
      OUT     D52.E  ; 異常 予備
692   LD      SM401  ; 常時OFF
      LD      T10  ; 制御電源 入 遅延
      AND     SM401  ; 常時OFF
      LD      D52.F  ; 異常 予備
      ANI     M2010  ; 異常リセット
      ORB
      ANB
      OUT     T147 K0  ; 異常 予備
      AND     T147  ; 異常 予備
      OUT     D52.F  ; 異常 予備
705   LD      SM400  ; 常時ON
      LD      T10  ; 制御電源 入 遅延
      AND     M37  ; 自動運転中まとめ
      AND     M1216  ; 搬入ﾌｫｰｸﾘﾌﾀ正転
      LD      D53.0  ; 搬入ﾌｫｰｸﾘﾌﾀ 上昇 ｻｲｸﾙｵｰﾊﾞｰ
      ANI     M2010  ; 異常リセット
      ORB
      ANB
      OUT     T148 D5101  ; 搬入ﾌｫｰｸﾘﾌﾀ 上昇 ｻｲｸﾙｵｰﾊﾞｰ 遅延 / ﾊﾟﾗﾒｰﾀ_搬入ﾌｫｰｸﾘﾌﾀ上昇ｻｲｸﾙｵｰﾊﾞｰ
      AND     T148  ; 搬入ﾌｫｰｸﾘﾌﾀ 上昇 ｻｲｸﾙｵｰﾊﾞｰ 遅延
      OUT     D53.0  ; 搬入ﾌｫｰｸﾘﾌﾀ 上昇 ｻｲｸﾙｵｰﾊﾞｰ
719   LD      SM400  ; 常時ON
      LD      T10  ; 制御電源 入 遅延
      AND     M37  ; 自動運転中まとめ
      AND     M1217  ; 搬入ﾌｫｰｸﾘﾌﾀ逆転
      LD      D53.1  ; 搬入ﾌｫｰｸﾘﾌﾀ 下降 ｻｲｸﾙｵｰﾊﾞｰ
      ANI     M2010  ; 異常リセット
      ORB
      ANB
      OUT     T149 D5102  ; 搬入ﾌｫｰｸﾘﾌﾀ 下降 ｻｲｸﾙｵｰﾊﾞｰ 遅延 / ﾊﾟﾗﾒｰﾀ_搬入ﾌｫｰｸﾘﾌﾀ下降ｻｲｸﾙｵｰﾊﾞｰ
      AND     T149  ; 搬入ﾌｫｰｸﾘﾌﾀ 下降 ｻｲｸﾙｵｰﾊﾞｰ 遅延
      OUT     D53.1  ; 搬入ﾌｫｰｸﾘﾌﾀ 下降 ｻｲｸﾙｵｰﾊﾞｰ
733   LD      SM400  ; 常時ON
      LD      T10  ; 制御電源 入 遅延
      LD      M30  ; 手動操作中
      OR      M37  ; 自動運転中まとめ
      ANB
      AND     M80  ; 搬入フォーク出 定位開始
      AND     M820  ; 搬入ﾌｫｰｸ_定位開始指令
      LD      D53.2  ; 搬入ﾌｫｰｸ 出 ｻｲｸﾙｵｰﾊﾞｰ
      ANI     M2010  ; 異常リセット
      ORB
      ANB
      OUT     T150 D5103  ; 搬入ﾌｫｰｸ 出 ｻｲｸﾙｵｰﾊﾞｰ 遅延 / ﾊﾟﾗﾒｰﾀ_搬入ﾌｫｰｸ 出 ｻｲｸﾙｵｰﾊﾞｰ
      AND     T150  ; 搬入ﾌｫｰｸ 出 ｻｲｸﾙｵｰﾊﾞｰ 遅延
      OUT     D53.2  ; 搬入ﾌｫｰｸ 出 ｻｲｸﾙｵｰﾊﾞｰ
750   LD      SM400  ; 常時ON
      LD      T10  ; 制御電源 入 遅延
      LD      M30  ; 手動操作中
      OR      M37  ; 自動運転中まとめ
      ANB
      AND     M81  ; 搬入フォーク戻 定位開始
      AND     M820  ; 搬入ﾌｫｰｸ_定位開始指令
      LD      D53.3  ; 搬入ﾌｫｰｸ 戻 ｻｲｸﾙｵｰﾊﾞｰ
      ANI     M2010  ; 異常リセット
      ORB
      ANB
      OUT     T151 D5104  ; 搬入ﾌｫｰｸ 戻 ｻｲｸﾙｵｰﾊﾞｰ 遅延 / ﾊﾟﾗﾒｰﾀ_搬入ﾌｫｰｸ 戻 ｻｲｸﾙｵｰﾊﾞｰ
      AND     T151  ; 搬入ﾌｫｰｸ 戻 ｻｲｸﾙｵｰﾊﾞｰ 遅延
      OUT     D53.3  ; 搬入ﾌｫｰｸ 戻 ｻｲｸﾙｵｰﾊﾞｰ
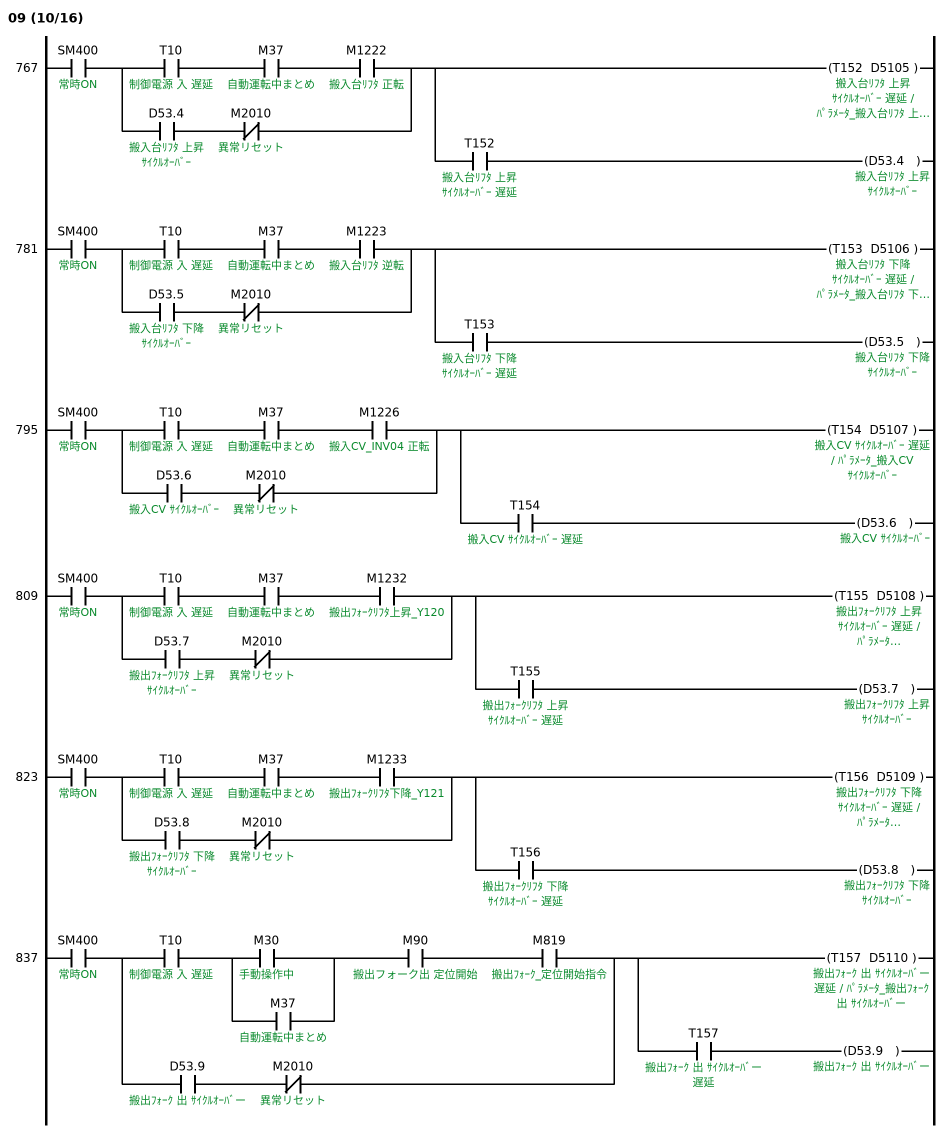
767   LD      SM400  ; 常時ON
      LD      T10  ; 制御電源 入 遅延
      AND     M37  ; 自動運転中まとめ
      AND     M1222  ; 搬入台ﾘﾌﾀ 正転
      LD      D53.4  ; 搬入台ﾘﾌﾀ 上昇 ｻｲｸﾙｵｰﾊﾞｰ
      ANI     M2010  ; 異常リセット
      ORB
      ANB
      OUT     T152 D5105  ; 搬入台ﾘﾌﾀ 上昇 ｻｲｸﾙｵｰﾊﾞｰ 遅延 / ﾊﾟﾗﾒｰﾀ_搬入台ﾘﾌﾀ 上昇 ｻｲｸﾙｵｰﾊﾞｰ
      AND     T152  ; 搬入台ﾘﾌﾀ 上昇 ｻｲｸﾙｵｰﾊﾞｰ 遅延
      OUT     D53.4  ; 搬入台ﾘﾌﾀ 上昇 ｻｲｸﾙｵｰﾊﾞｰ
781   LD      SM400  ; 常時ON
      LD      T10  ; 制御電源 入 遅延
      AND     M37  ; 自動運転中まとめ
      AND     M1223  ; 搬入台ﾘﾌﾀ 逆転
      LD      D53.5  ; 搬入台ﾘﾌﾀ 下降 ｻｲｸﾙｵｰﾊﾞｰ
      ANI     M2010  ; 異常リセット
      ORB
      ANB
      OUT     T153 D5106  ; 搬入台ﾘﾌﾀ 下降 ｻｲｸﾙｵｰﾊﾞｰ 遅延 / ﾊﾟﾗﾒｰﾀ_搬入台ﾘﾌﾀ 下降 ｻｲｸﾙｵｰﾊﾞｰ
      AND     T153  ; 搬入台ﾘﾌﾀ 下降 ｻｲｸﾙｵｰﾊﾞｰ 遅延
      OUT     D53.5  ; 搬入台ﾘﾌﾀ 下降 ｻｲｸﾙｵｰﾊﾞｰ
795   LD      SM400  ; 常時ON
      LD      T10  ; 制御電源 入 遅延
      AND     M37  ; 自動運転中まとめ
      AND     M1226  ; 搬入CV_INV04 正転
      LD      D53.6  ; 搬入CV ｻｲｸﾙｵｰﾊﾞｰ
      ANI     M2010  ; 異常リセット
      ORB
      ANB
      OUT     T154 D5107  ; 搬入CV ｻｲｸﾙｵｰﾊﾞｰ 遅延 / ﾊﾟﾗﾒｰﾀ_搬入CV ｻｲｸﾙｵｰﾊﾞｰ
      AND     T154  ; 搬入CV ｻｲｸﾙｵｰﾊﾞｰ 遅延
      OUT     D53.6  ; 搬入CV ｻｲｸﾙｵｰﾊﾞｰ
809   LD      SM400  ; 常時ON
      LD      T10  ; 制御電源 入 遅延
      AND     M37  ; 自動運転中まとめ
      AND     M1232  ; 搬出ﾌｫｰｸﾘﾌﾀ上昇_Y120
      LD      D53.7  ; 搬出ﾌｫｰｸﾘﾌﾀ 上昇 ｻｲｸﾙｵｰﾊﾞｰ
      ANI     M2010  ; 異常リセット
      ORB
      ANB
      OUT     T155 D5108  ; 搬出ﾌｫｰｸﾘﾌﾀ 上昇 ｻｲｸﾙｵｰﾊﾞｰ 遅延 / ﾊﾟﾗﾒｰﾀ_搬出ﾌｫｰｸﾘﾌﾀ上昇ｻｲｸﾙｵｰﾊﾞｰ
      AND     T155  ; 搬出ﾌｫｰｸﾘﾌﾀ 上昇 ｻｲｸﾙｵｰﾊﾞｰ 遅延
      OUT     D53.7  ; 搬出ﾌｫｰｸﾘﾌﾀ 上昇 ｻｲｸﾙｵｰﾊﾞｰ
823   LD      SM400  ; 常時ON
      LD      T10  ; 制御電源 入 遅延
      AND     M37  ; 自動運転中まとめ
      AND     M1233  ; 搬出ﾌｫｰｸﾘﾌﾀ下降_Y121
      LD      D53.8  ; 搬出ﾌｫｰｸﾘﾌﾀ 下降 ｻｲｸﾙｵｰﾊﾞｰ
      ANI     M2010  ; 異常リセット
      ORB
      ANB
      OUT     T156 D5109  ; 搬出ﾌｫｰｸﾘﾌﾀ 下降 ｻｲｸﾙｵｰﾊﾞｰ 遅延 / ﾊﾟﾗﾒｰﾀ_搬出ﾌｫｰｸﾘﾌﾀ下降ｻｲｸﾙｵｰﾊﾞｰ
      AND     T156  ; 搬出ﾌｫｰｸﾘﾌﾀ 下降 ｻｲｸﾙｵｰﾊﾞｰ 遅延
      OUT     D53.8  ; 搬出ﾌｫｰｸﾘﾌﾀ 下降 ｻｲｸﾙｵｰﾊﾞｰ
837   LD      SM400  ; 常時ON
      LD      T10  ; 制御電源 入 遅延
      LD      M30  ; 手動操作中
      OR      M37  ; 自動運転中まとめ
      ANB
      AND     M90  ; 搬出フォーク出 定位開始
      AND     M819  ; 搬出ﾌｫｰｸ_定位開始指令
      LD      D53.9  ; 搬出ﾌｫｰｸ 出 ｻｲｸﾙｵｰﾊﾞー
      ANI     M2010  ; 異常リセット
      ORB
      ANB
      OUT     T157 D5110  ; 搬出ﾌｫｰｸ 出 ｻｲｸﾙｵｰﾊﾞー 遅延 / ﾊﾟﾗﾒｰﾀ_搬出ﾌｫｰｸ 出 ｻｲｸﾙｵｰﾊﾞー
      AND     T157  ; 搬出ﾌｫｰｸ 出 ｻｲｸﾙｵｰﾊﾞー 遅延
      OUT     D53.9  ; 搬出ﾌｫｰｸ 出 ｻｲｸﾙｵｰﾊﾞー
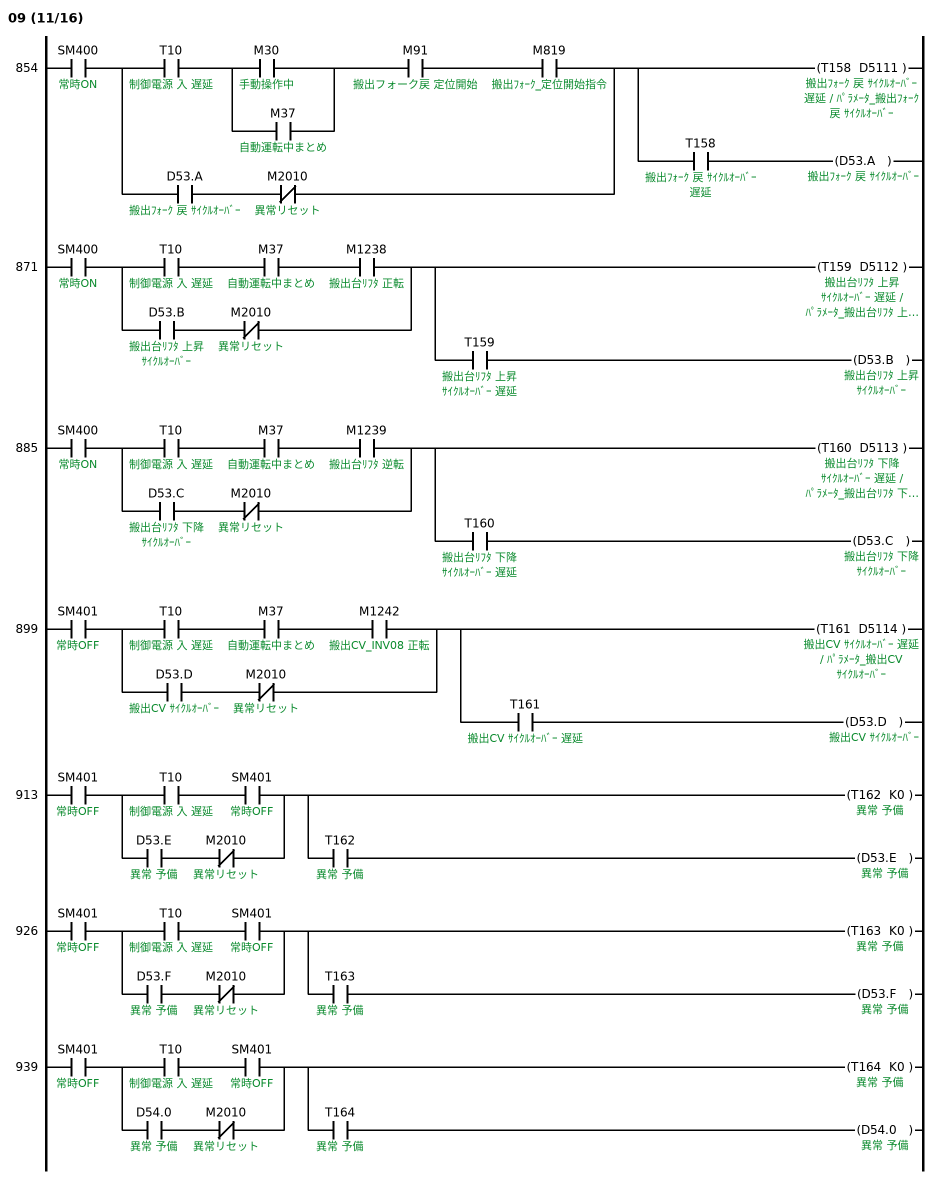
854   LD      SM400  ; 常時ON
      LD      T10  ; 制御電源 入 遅延
      LD      M30  ; 手動操作中
      OR      M37  ; 自動運転中まとめ
      ANB
      AND     M91  ; 搬出フォーク戻 定位開始
      AND     M819  ; 搬出ﾌｫｰｸ_定位開始指令
      LD      D53.A  ; 搬出ﾌｫｰｸ 戻 ｻｲｸﾙｵｰﾊﾞｰ
      ANI     M2010  ; 異常リセット
      ORB
      ANB
      OUT     T158 D5111  ; 搬出ﾌｫｰｸ 戻 ｻｲｸﾙｵｰﾊﾞｰ 遅延 / ﾊﾟﾗﾒｰﾀ_搬出ﾌｫｰｸ 戻 ｻｲｸﾙｵｰﾊﾞｰ
      AND     T158  ; 搬出ﾌｫｰｸ 戻 ｻｲｸﾙｵｰﾊﾞｰ 遅延
      OUT     D53.A  ; 搬出ﾌｫｰｸ 戻 ｻｲｸﾙｵｰﾊﾞｰ
871   LD      SM400  ; 常時ON
      LD      T10  ; 制御電源 入 遅延
      AND     M37  ; 自動運転中まとめ
      AND     M1238  ; 搬出台ﾘﾌﾀ 正転
      LD      D53.B  ; 搬出台ﾘﾌﾀ 上昇 ｻｲｸﾙｵｰﾊﾞｰ
      ANI     M2010  ; 異常リセット
      ORB
      ANB
      OUT     T159 D5112  ; 搬出台ﾘﾌﾀ 上昇 ｻｲｸﾙｵｰﾊﾞｰ 遅延 / ﾊﾟﾗﾒｰﾀ_搬出台ﾘﾌﾀ 上昇 ｻｲｸﾙｵｰﾊﾞｰ
      AND     T159  ; 搬出台ﾘﾌﾀ 上昇 ｻｲｸﾙｵｰﾊﾞｰ 遅延
      OUT     D53.B  ; 搬出台ﾘﾌﾀ 上昇 ｻｲｸﾙｵｰﾊﾞｰ
885   LD      SM400  ; 常時ON
      LD      T10  ; 制御電源 入 遅延
      AND     M37  ; 自動運転中まとめ
      AND     M1239  ; 搬出台ﾘﾌﾀ 逆転
      LD      D53.C  ; 搬出台ﾘﾌﾀ 下降 ｻｲｸﾙｵｰﾊﾞｰ
      ANI     M2010  ; 異常リセット
      ORB
      ANB
      OUT     T160 D5113  ; 搬出台ﾘﾌﾀ 下降 ｻｲｸﾙｵｰﾊﾞｰ 遅延 / ﾊﾟﾗﾒｰﾀ_搬出台ﾘﾌﾀ 下降 ｻｲｸﾙｵｰﾊﾞｰ
      AND     T160  ; 搬出台ﾘﾌﾀ 下降 ｻｲｸﾙｵｰﾊﾞｰ 遅延
      OUT     D53.C  ; 搬出台ﾘﾌﾀ 下降 ｻｲｸﾙｵｰﾊﾞｰ
899   LD      SM401  ; 常時OFF
      LD      T10  ; 制御電源 入 遅延
      AND     M37  ; 自動運転中まとめ
      AND     M1242  ; 搬出CV_INV08 正転
      LD      D53.D  ; 搬出CV ｻｲｸﾙｵｰﾊﾞｰ
      ANI     M2010  ; 異常リセット
      ORB
      ANB
      OUT     T161 D5114  ; 搬出CV ｻｲｸﾙｵｰﾊﾞｰ 遅延 / ﾊﾟﾗﾒｰﾀ_搬出CV ｻｲｸﾙｵｰﾊﾞｰ
      AND     T161  ; 搬出CV ｻｲｸﾙｵｰﾊﾞｰ 遅延
      OUT     D53.D  ; 搬出CV ｻｲｸﾙｵｰﾊﾞｰ
913   LD      SM401  ; 常時OFF
      LD      T10  ; 制御電源 入 遅延
      AND     SM401  ; 常時OFF
      LD      D53.E  ; 異常 予備
      ANI     M2010  ; 異常リセット
      ORB
      ANB
      OUT     T162 K0  ; 異常 予備
      AND     T162  ; 異常 予備
      OUT     D53.E  ; 異常 予備
926   LD      SM401  ; 常時OFF
      LD      T10  ; 制御電源 入 遅延
      AND     SM401  ; 常時OFF
      LD      D53.F  ; 異常 予備
      ANI     M2010  ; 異常リセット
      ORB
      ANB
      OUT     T163 K0  ; 異常 予備
      AND     T163  ; 異常 予備
      OUT     D53.F  ; 異常 予備
939   LD      SM401  ; 常時OFF
      LD      T10  ; 制御電源 入 遅延
      AND     SM401  ; 常時OFF
      LD      D54.0  ; 異常 予備
      ANI     M2010  ; 異常リセット
      ORB
      ANB
      OUT     T164 K0  ; 異常 予備
      AND     T164  ; 異常 予備
      OUT     D54.0  ; 異常 予備
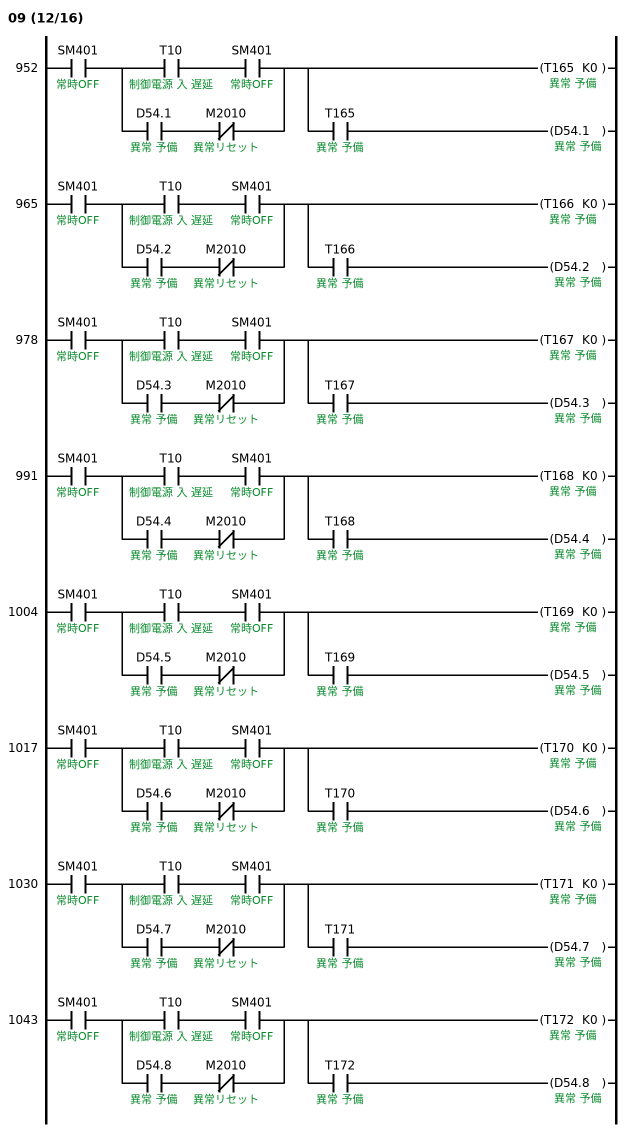
952   LD      SM401  ; 常時OFF
      LD      T10  ; 制御電源 入 遅延
      AND     SM401  ; 常時OFF
      LD      D54.1  ; 異常 予備
      ANI     M2010  ; 異常リセット
      ORB
      ANB
      OUT     T165 K0  ; 異常 予備
      AND     T165  ; 異常 予備
      OUT     D54.1  ; 異常 予備
965   LD      SM401  ; 常時OFF
      LD      T10  ; 制御電源 入 遅延
      AND     SM401  ; 常時OFF
      LD      D54.2  ; 異常 予備
      ANI     M2010  ; 異常リセット
      ORB
      ANB
      OUT     T166 K0  ; 異常 予備
      AND     T166  ; 異常 予備
      OUT     D54.2  ; 異常 予備
978   LD      SM401  ; 常時OFF
      LD      T10  ; 制御電源 入 遅延
      AND     SM401  ; 常時OFF
      LD      D54.3  ; 異常 予備
      ANI     M2010  ; 異常リセット
      ORB
      ANB
      OUT     T167 K0  ; 異常 予備
      AND     T167  ; 異常 予備
      OUT     D54.3  ; 異常 予備
991   LD      SM401  ; 常時OFF
      LD      T10  ; 制御電源 入 遅延
      AND     SM401  ; 常時OFF
      LD      D54.4  ; 異常 予備
      ANI     M2010  ; 異常リセット
      ORB
      ANB
      OUT     T168 K0  ; 異常 予備
      AND     T168  ; 異常 予備
      OUT     D54.4  ; 異常 予備
1004  LD      SM401  ; 常時OFF
      LD      T10  ; 制御電源 入 遅延
      AND     SM401  ; 常時OFF
      LD      D54.5  ; 異常 予備
      ANI     M2010  ; 異常リセット
      ORB
      ANB
      OUT     T169 K0  ; 異常 予備
      AND     T169  ; 異常 予備
      OUT     D54.5  ; 異常 予備
1017  LD      SM401  ; 常時OFF
      LD      T10  ; 制御電源 入 遅延
      AND     SM401  ; 常時OFF
      LD      D54.6  ; 異常 予備
      ANI     M2010  ; 異常リセット
      ORB
      ANB
      OUT     T170 K0  ; 異常 予備
      AND     T170  ; 異常 予備
      OUT     D54.6  ; 異常 予備
1030  LD      SM401  ; 常時OFF
      LD      T10  ; 制御電源 入 遅延
      AND     SM401  ; 常時OFF
      LD      D54.7  ; 異常 予備
      ANI     M2010  ; 異常リセット
      ORB
      ANB
      OUT     T171 K0  ; 異常 予備
      AND     T171  ; 異常 予備
      OUT     D54.7  ; 異常 予備
1043  LD      SM401  ; 常時OFF
      LD      T10  ; 制御電源 入 遅延
      AND     SM401  ; 常時OFF
      LD      D54.8  ; 異常 予備
      ANI     M2010  ; 異常リセット
      ORB
      ANB
      OUT     T172 K0  ; 異常 予備
      AND     T172  ; 異常 予備
      OUT     D54.8  ; 異常 予備
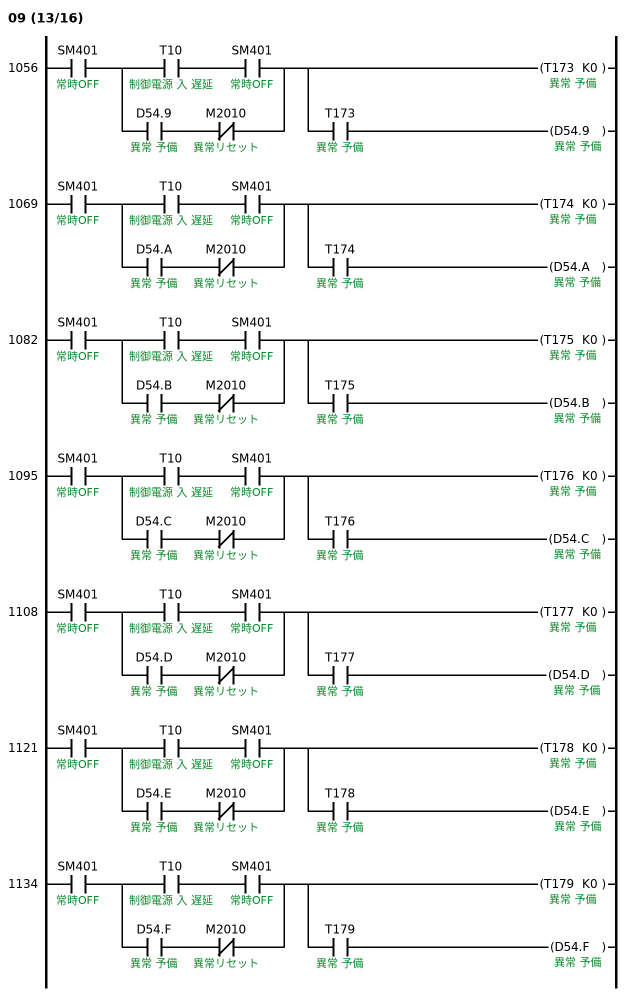
1056  LD      SM401  ; 常時OFF
      LD      T10  ; 制御電源 入 遅延
      AND     SM401  ; 常時OFF
      LD      D54.9  ; 異常 予備
      ANI     M2010  ; 異常リセット
      ORB
      ANB
      OUT     T173 K0  ; 異常 予備
      AND     T173  ; 異常 予備
      OUT     D54.9  ; 異常 予備
1069  LD      SM401  ; 常時OFF
      LD      T10  ; 制御電源 入 遅延
      AND     SM401  ; 常時OFF
      LD      D54.A  ; 異常 予備
      ANI     M2010  ; 異常リセット
      ORB
      ANB
      OUT     T174 K0  ; 異常 予備
      AND     T174  ; 異常 予備
      OUT     D54.A  ; 異常 予備
1082  LD      SM401  ; 常時OFF
      LD      T10  ; 制御電源 入 遅延
      AND     SM401  ; 常時OFF
      LD      D54.B  ; 異常 予備
      ANI     M2010  ; 異常リセット
      ORB
      ANB
      OUT     T175 K0  ; 異常 予備
      AND     T175  ; 異常 予備
      OUT     D54.B  ; 異常 予備
1095  LD      SM401  ; 常時OFF
      LD      T10  ; 制御電源 入 遅延
      AND     SM401  ; 常時OFF
      LD      D54.C  ; 異常 予備
      ANI     M2010  ; 異常リセット
      ORB
      ANB
      OUT     T176 K0  ; 異常 予備
      AND     T176  ; 異常 予備
      OUT     D54.C  ; 異常 予備
1108  LD      SM401  ; 常時OFF
      LD      T10  ; 制御電源 入 遅延
      AND     SM401  ; 常時OFF
      LD      D54.D  ; 異常 予備
      ANI     M2010  ; 異常リセット
      ORB
      ANB
      OUT     T177 K0  ; 異常 予備
      AND     T177  ; 異常 予備
      OUT     D54.D  ; 異常 予備
1121  LD      SM401  ; 常時OFF
      LD      T10  ; 制御電源 入 遅延
      AND     SM401  ; 常時OFF
      LD      D54.E  ; 異常 予備
      ANI     M2010  ; 異常リセット
      ORB
      ANB
      OUT     T178 K0  ; 異常 予備
      AND     T178  ; 異常 予備
      OUT     D54.E  ; 異常 予備
1134  LD      SM401  ; 常時OFF
      LD      T10  ; 制御電源 入 遅延
      AND     SM401  ; 常時OFF
      LD      D54.F  ; 異常 予備
      ANI     M2010  ; 異常リセット
      ORB
      ANB
      OUT     T179 K0  ; 異常 予備
      AND     T179  ; 異常 予備
      OUT     D54.F  ; 異常 予備
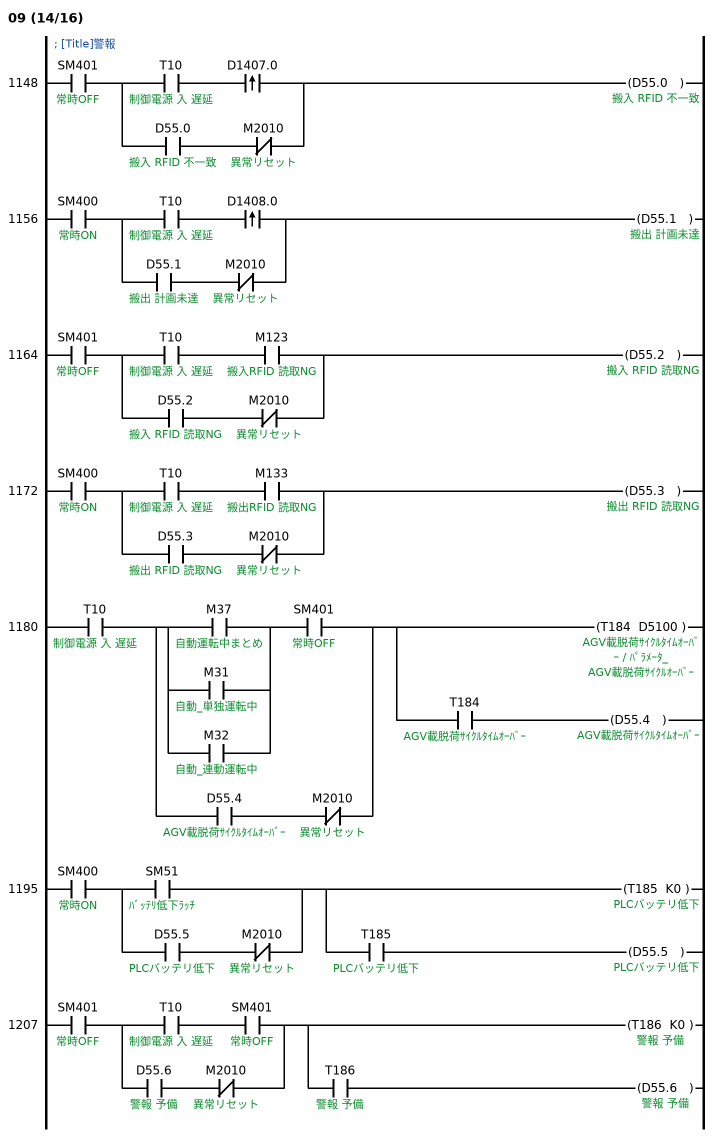
; [Title]警報
1148  LD      SM401  ; 常時OFF
      LD      T10  ; 制御電源 入 遅延
      ANDP    D1407.0
      LD      D55.0  ; 搬入 RFID 不一致
      ANI     M2010  ; 異常リセット
      ORB
      ANB
      OUT     D55.0  ; 搬入 RFID 不一致
1156  LD      SM400  ; 常時ON
      LD      T10  ; 制御電源 入 遅延
      ANDP    D1408.0
      LD      D55.1  ; 搬出 計画未達
      ANI     M2010  ; 異常リセット
      ORB
      ANB
      OUT     D55.1  ; 搬出 計画未達
1164  LD      SM401  ; 常時OFF
      LD      T10  ; 制御電源 入 遅延
      AND     M123  ; 搬入RFID 読取NG
      LD      D55.2  ; 搬入 RFID 読取NG
      ANI     M2010  ; 異常リセット
      ORB
      ANB
      OUT     D55.2  ; 搬入 RFID 読取NG
1172  LD      SM400  ; 常時ON
      LD      T10  ; 制御電源 入 遅延
      AND     M133  ; 搬出RFID 読取NG
      LD      D55.3  ; 搬出 RFID 読取NG
      ANI     M2010  ; 異常リセット
      ORB
      ANB
      OUT     D55.3  ; 搬出 RFID 読取NG
1180  LD      T10  ; 制御電源 入 遅延
      LD      M37  ; 自動運転中まとめ
      OR      M31  ; 自動_単独運転中
      OR      M32  ; 自動_連動運転中
      AND     SM401  ; 常時OFF
      LD      D55.4  ; AGV載脱荷ｻｲｸﾙﾀｲﾑｵｰﾊﾞｰ
      ANI     M2010  ; 異常リセット
      ORB
      ANB
      OUT     T184 D5100  ; AGV載脱荷ｻｲｸﾙﾀｲﾑｵｰﾊﾞｰ / ﾊﾟﾗﾒｰﾀ_AGV載脱荷ｻｲｸﾙｵｰﾊﾞｰ
      AND     T184  ; AGV載脱荷ｻｲｸﾙﾀｲﾑｵｰﾊﾞｰ
      OUT     D55.4  ; AGV載脱荷ｻｲｸﾙﾀｲﾑｵｰﾊﾞｰ
1195  LD      SM400  ; 常時ON
      LD      SM51  ; ﾊﾞｯﾃﾘ低下ﾗｯﾁ
      LD      D55.5  ; PLCバッテリ低下
      ANI     M2010  ; 異常リセット
      ORB
      ANB
      OUT     T185 K0  ; PLCバッテリ低下
      AND     T185  ; PLCバッテリ低下
      OUT     D55.5  ; PLCバッテリ低下
1207  LD      SM401  ; 常時OFF
      LD      T10  ; 制御電源 入 遅延
      AND     SM401  ; 常時OFF
      LD      D55.6  ; 警報 予備
      ANI     M2010  ; 異常リセット
      ORB
      ANB
      OUT     T186 K0  ; 警報 予備
      AND     T186  ; 警報 予備
      OUT     D55.6  ; 警報 予備
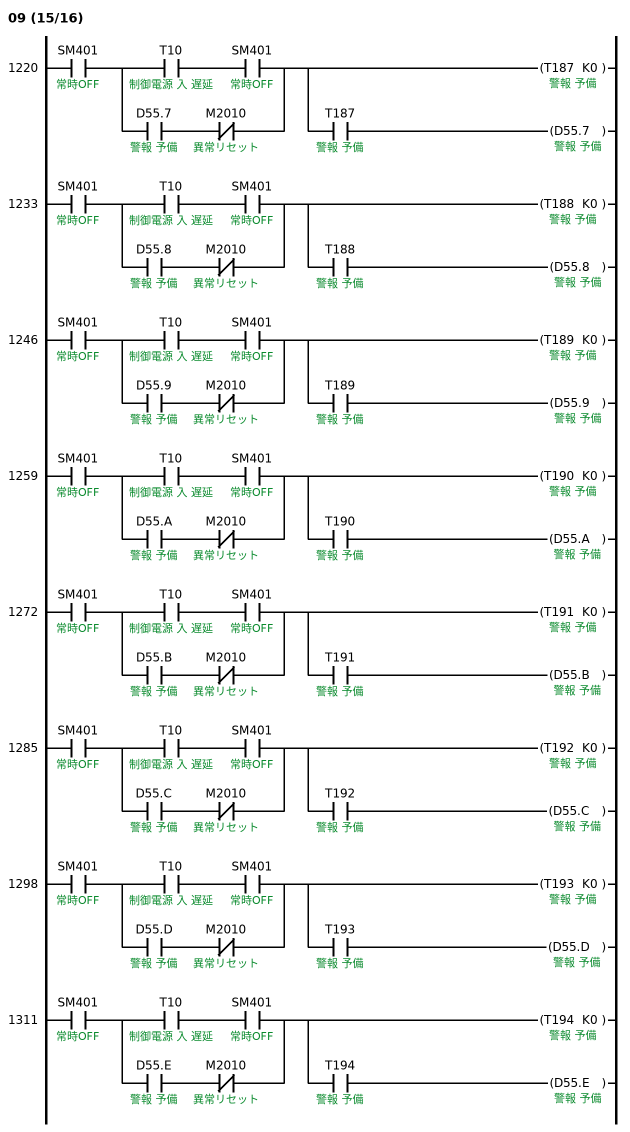
1220  LD      SM401  ; 常時OFF
      LD      T10  ; 制御電源 入 遅延
      AND     SM401  ; 常時OFF
      LD      D55.7  ; 警報 予備
      ANI     M2010  ; 異常リセット
      ORB
      ANB
      OUT     T187 K0  ; 警報 予備
      AND     T187  ; 警報 予備
      OUT     D55.7  ; 警報 予備
1233  LD      SM401  ; 常時OFF
      LD      T10  ; 制御電源 入 遅延
      AND     SM401  ; 常時OFF
      LD      D55.8  ; 警報 予備
      ANI     M2010  ; 異常リセット
      ORB
      ANB
      OUT     T188 K0  ; 警報 予備
      AND     T188  ; 警報 予備
      OUT     D55.8  ; 警報 予備
1246  LD      SM401  ; 常時OFF
      LD      T10  ; 制御電源 入 遅延
      AND     SM401  ; 常時OFF
      LD      D55.9  ; 警報 予備
      ANI     M2010  ; 異常リセット
      ORB
      ANB
      OUT     T189 K0  ; 警報 予備
      AND     T189  ; 警報 予備
      OUT     D55.9  ; 警報 予備
1259  LD      SM401  ; 常時OFF
      LD      T10  ; 制御電源 入 遅延
      AND     SM401  ; 常時OFF
      LD      D55.A  ; 警報 予備
      ANI     M2010  ; 異常リセット
      ORB
      ANB
      OUT     T190 K0  ; 警報 予備
      AND     T190  ; 警報 予備
      OUT     D55.A  ; 警報 予備
1272  LD      SM401  ; 常時OFF
      LD      T10  ; 制御電源 入 遅延
      AND     SM401  ; 常時OFF
      LD      D55.B  ; 警報 予備
      ANI     M2010  ; 異常リセット
      ORB
      ANB
      OUT     T191 K0  ; 警報 予備
      AND     T191  ; 警報 予備
      OUT     D55.B  ; 警報 予備
1285  LD      SM401  ; 常時OFF
      LD      T10  ; 制御電源 入 遅延
      AND     SM401  ; 常時OFF
      LD      D55.C  ; 警報 予備
      ANI     M2010  ; 異常リセット
      ORB
      ANB
      OUT     T192 K0  ; 警報 予備
      AND     T192  ; 警報 予備
      OUT     D55.C  ; 警報 予備
1298  LD      SM401  ; 常時OFF
      LD      T10  ; 制御電源 入 遅延
      AND     SM401  ; 常時OFF
      LD      D55.D  ; 警報 予備
      ANI     M2010  ; 異常リセット
      ORB
      ANB
      OUT     T193 K0  ; 警報 予備
      AND     T193  ; 警報 予備
      OUT     D55.D  ; 警報 予備
1311  LD      SM401  ; 常時OFF
      LD      T10  ; 制御電源 入 遅延
      AND     SM401  ; 常時OFF
      LD      D55.E  ; 警報 予備
      ANI     M2010  ; 異常リセット
      ORB
      ANB
      OUT     T194 K0  ; 警報 予備
      AND     T194  ; 警報 予備
      OUT     D55.E  ; 警報 予備
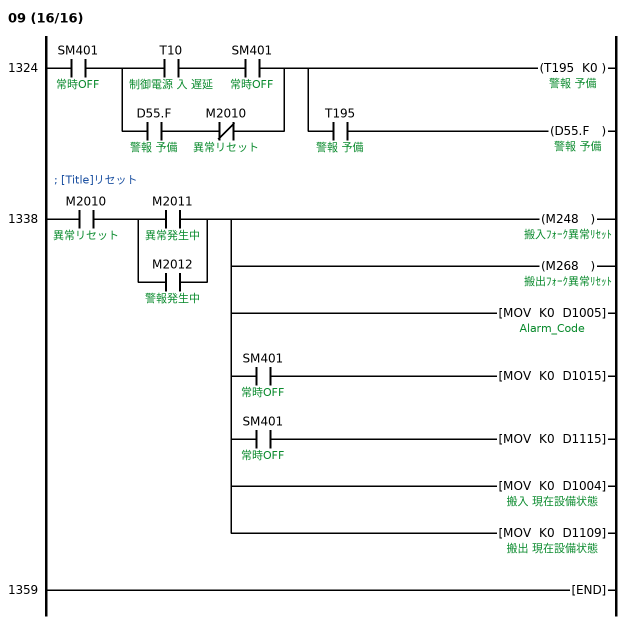
1324  LD      SM401  ; 常時OFF
      LD      T10  ; 制御電源 入 遅延
      AND     SM401  ; 常時OFF
      LD      D55.F  ; 警報 予備
      ANI     M2010  ; 異常リセット
      ORB
      ANB
      OUT     T195 K0  ; 警報 予備
      AND     T195  ; 警報 予備
      OUT     D55.F  ; 警報 予備
; [Title]リセット
1338  LD      M2010  ; 異常リセット
      LD      M2011  ; 異常発生中
      OR      M2012  ; 警報発生中
      ANB
      OUT     M248  ; 搬入ﾌｫｰｸ異常ﾘｾｯﾄ
      OUT     M268  ; 搬出ﾌｫｰｸ異常ﾘｾｯﾄ
      MOV     K0 D1005  ; Alarm_Code
      MPS
      AND     SM401  ; 常時OFF
      MOV     K0 D1015
      MRD
      AND     SM401  ; 常時OFF
      MOV     K0 D1115
      MPP
      MOV     K0 D1004
      MOV     K0 D1109
1359  END
END_PROGRAM

PROGRAM 10  // MAIN
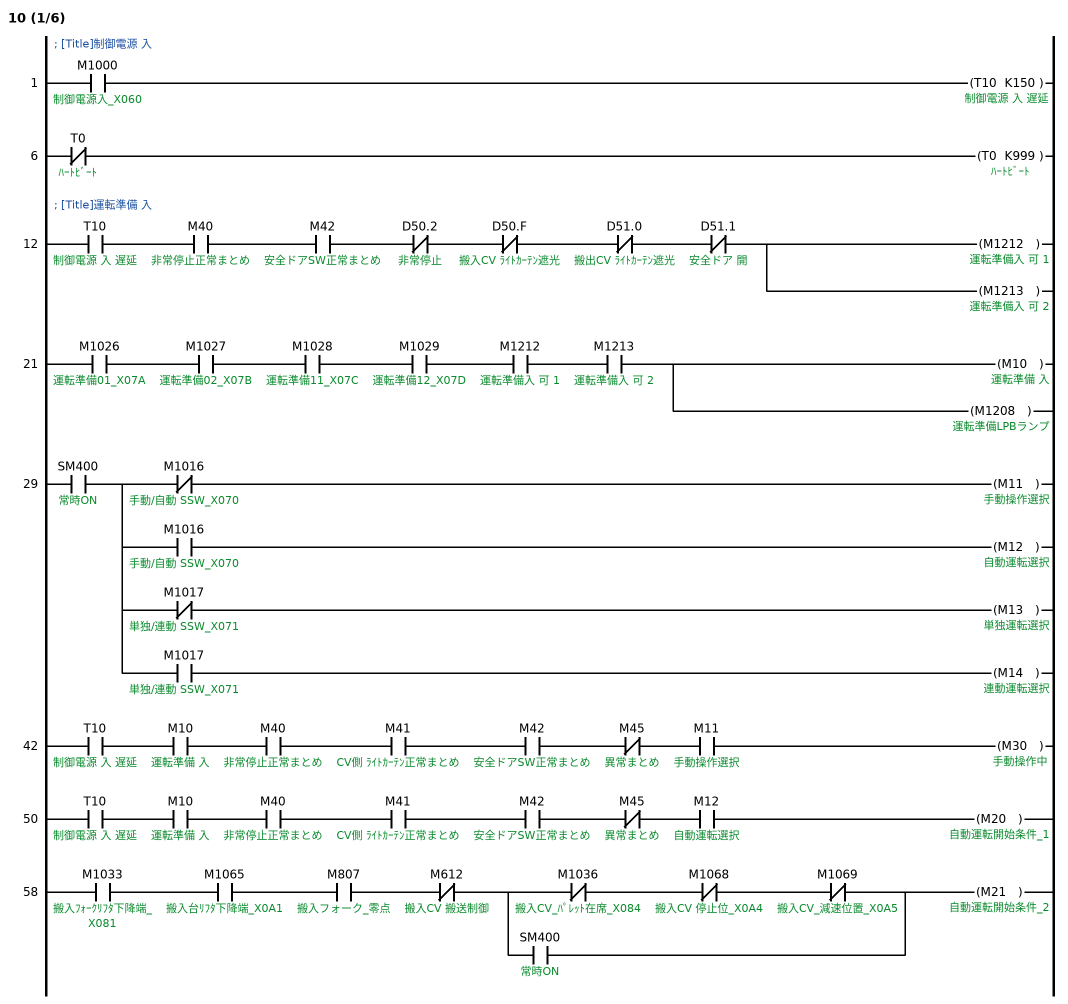
; [Title]制御電源 入
1     LD      M1000  ; 制御電源入_X060
      OUT     T10 K150  ; 制御電源 入 遅延
6     LDI     T0  ; ﾊｰﾄﾋﾞｰﾄ
      OUT     T0 K999  ; ﾊｰﾄﾋﾞｰﾄ
; [Title]運転準備 入
12    LD      T10  ; 制御電源 入 遅延
      AND     M40  ; 非常停止正常まとめ
      AND     M42  ; 安全ドアSW正常まとめ
      ANI     D50.2  ; 非常停止
      ANI     D50.F  ; 搬入CV ﾗｲﾄｶｰﾃﾝ遮光
      ANI     D51.0  ; 搬出CV ﾗｲﾄｶｰﾃﾝ遮光
      ANI     D51.1  ; 安全ドア 開
      OUT     M1212  ; 運転準備入 可 1
      OUT     M1213  ; 運転準備入 可 2
21    LD      M1026  ; 運転準備01_X07A
      AND     M1027  ; 運転準備02_X07B
      AND     M1028  ; 運転準備11_X07C
      AND     M1029  ; 運転準備12_X07D
      AND     M1212  ; 運転準備入 可 1
      AND     M1213  ; 運転準備入 可 2
      OUT     M10  ; 運転準備 入
      OUT     M1208  ; 運転準備LPBランプ
29    LD      SM400  ; 常時ON
      MPS
      ANI     M1016  ; 手動/自動 SSW_X070
      OUT     M11  ; 手動操作選択
      MRD
      AND     M1016  ; 手動/自動 SSW_X070
      OUT     M12  ; 自動運転選択
      MRD
      ANI     M1017  ; 単独/連動 SSW_X071
      OUT     M13  ; 単独運転選択
      MPP
      AND     M1017  ; 単独/連動 SSW_X071
      OUT     M14  ; 連動運転選択
42    LD      T10  ; 制御電源 入 遅延
      AND     M10  ; 運転準備 入
      AND     M40  ; 非常停止正常まとめ
      AND     M41  ; CV側 ﾗｲﾄｶｰﾃﾝ正常まとめ
      AND     M42  ; 安全ドアSW正常まとめ
      ANI     M45  ; 異常まとめ
      AND     M11  ; 手動操作選択
      OUT     M30  ; 手動操作中
50    LD      T10  ; 制御電源 入 遅延
      AND     M10  ; 運転準備 入
      AND     M40  ; 非常停止正常まとめ
      AND     M41  ; CV側 ﾗｲﾄｶｰﾃﾝ正常まとめ
      AND     M42  ; 安全ドアSW正常まとめ
      ANI     M45  ; 異常まとめ
      AND     M12  ; 自動運転選択
      OUT     M20  ; 自動運転開始条件_1
58    LD      M1033  ; 搬入ﾌｫｰｸﾘﾌﾀ下降端_X081
      AND     M1065  ; 搬入台ﾘﾌﾀ下降端_X0A1
      AND     M807  ; 搬入フォーク_零点
      ANI     M612  ; 搬入CV 搬送制御
      LDI     M1036  ; 搬入CV_ﾊﾟﾚｯﾄ在席_X084
      ANI     M1068  ; 搬入CV 停止位_X0A4
      ANI     M1069  ; 搬入CV_減速位置_X0A5
      OR      SM400  ; 常時ON
      ANB
      OUT     M21  ; 自動運転開始条件_2
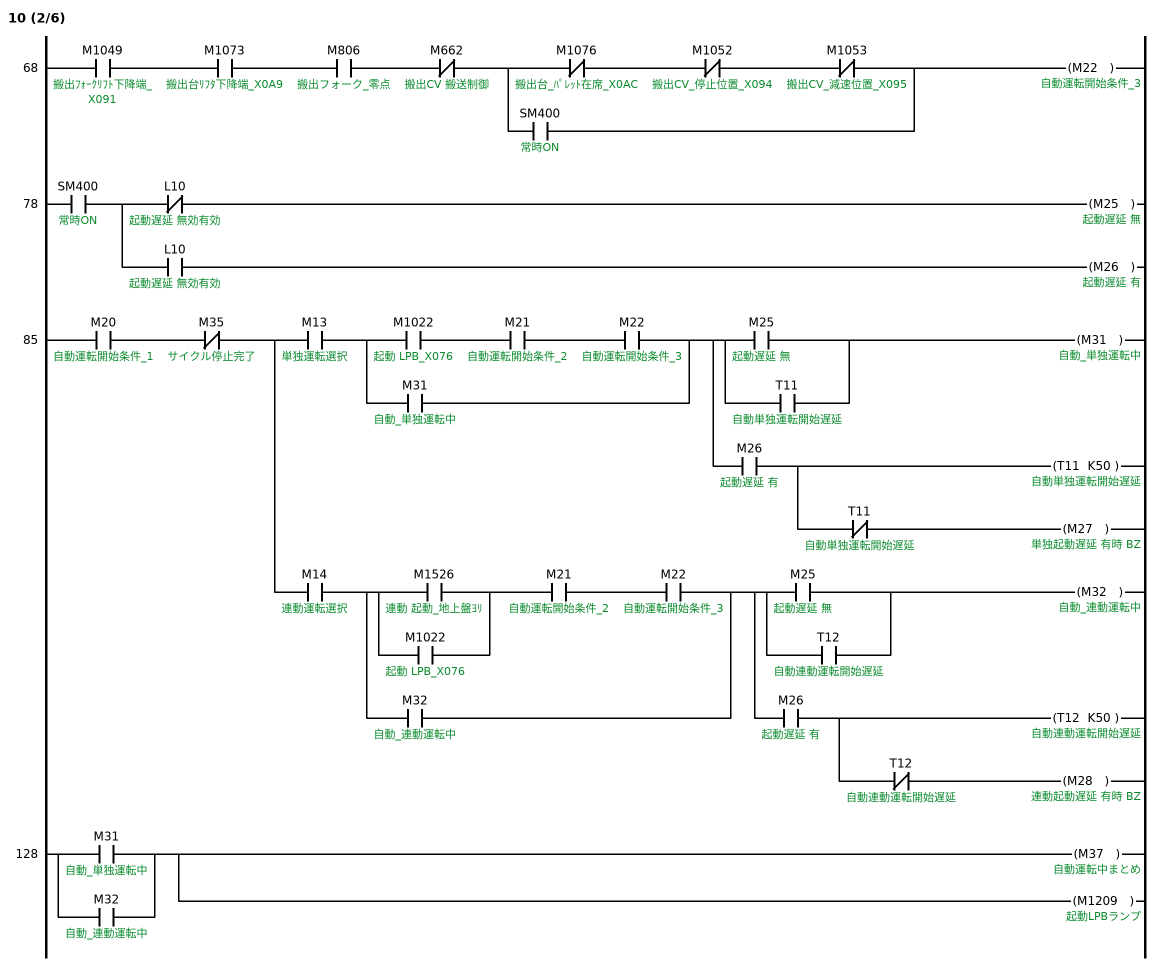
68    LD      M1049  ; 搬出ﾌｫｰｸﾘﾌﾄ下降端_X091
      AND     M1073  ; 搬出台ﾘﾌﾀ下降端_X0A9
      AND     M806  ; 搬出フォーク_零点
      ANI     M662  ; 搬出CV 搬送制御
      LDI     M1076  ; 搬出台_ﾊﾟﾚｯﾄ在席_X0AC
      ANI     M1052  ; 搬出CV_停止位置_X094
      ANI     M1053  ; 搬出CV_減速位置_X095
      OR      SM400  ; 常時ON
      ANB
      OUT     M22  ; 自動運転開始条件_3
78    LD      SM400  ; 常時ON
      MPS
      ANI     L10  ; 起動遅延 無効有効
      OUT     M25  ; 起動遅延 無
      MPP
      AND     L10  ; 起動遅延 無効有効
      OUT     M26  ; 起動遅延 有
85    LD      M20  ; 自動運転開始条件_1
      ANI     M35  ; サイクル停止完了
      MPS
      AND     M13  ; 単独運転選択
      LD      M1022  ; 起動 LPB_X076
      AND     M21  ; 自動運転開始条件_2
      AND     M22  ; 自動運転開始条件_3
      OR      M31  ; 自動_単独運転中
      ANB
      MPS
      LD      M25  ; 起動遅延 無
      OR      T11  ; 自動単独運転開始遅延
      ANB
      OUT     M31  ; 自動_単独運転中
      MPP
      AND     M26  ; 起動遅延 有
      OUT     T11 K50  ; 自動単独運転開始遅延
      ANI     T11  ; 自動単独運転開始遅延
      OUT     M27  ; 単独起動遅延 有時 BZ
      MPP
      AND     M14  ; 連動運転選択
      LD      M1526  ; 連動 起動_地上盤ﾖﾘ
      OR      M1022  ; 起動 LPB_X076
      AND     M21  ; 自動運転開始条件_2
      AND     M22  ; 自動運転開始条件_3
      OR      M32  ; 自動_連動運転中
      ANB
      MPS
      LD      M25  ; 起動遅延 無
      OR      T12  ; 自動連動運転開始遅延
      ANB
      OUT     M32  ; 自動_連動運転中
      MPP
      AND     M26  ; 起動遅延 有
      OUT     T12 K50  ; 自動連動運転開始遅延
      ANI     T12  ; 自動連動運転開始遅延
      OUT     M28  ; 連動起動遅延 有時 BZ
128   LD      M31  ; 自動_単独運転中
      OR      M32  ; 自動_連動運転中
      OUT     M37  ; 自動運転中まとめ
      OUT     M1209  ; 起動LPBランプ
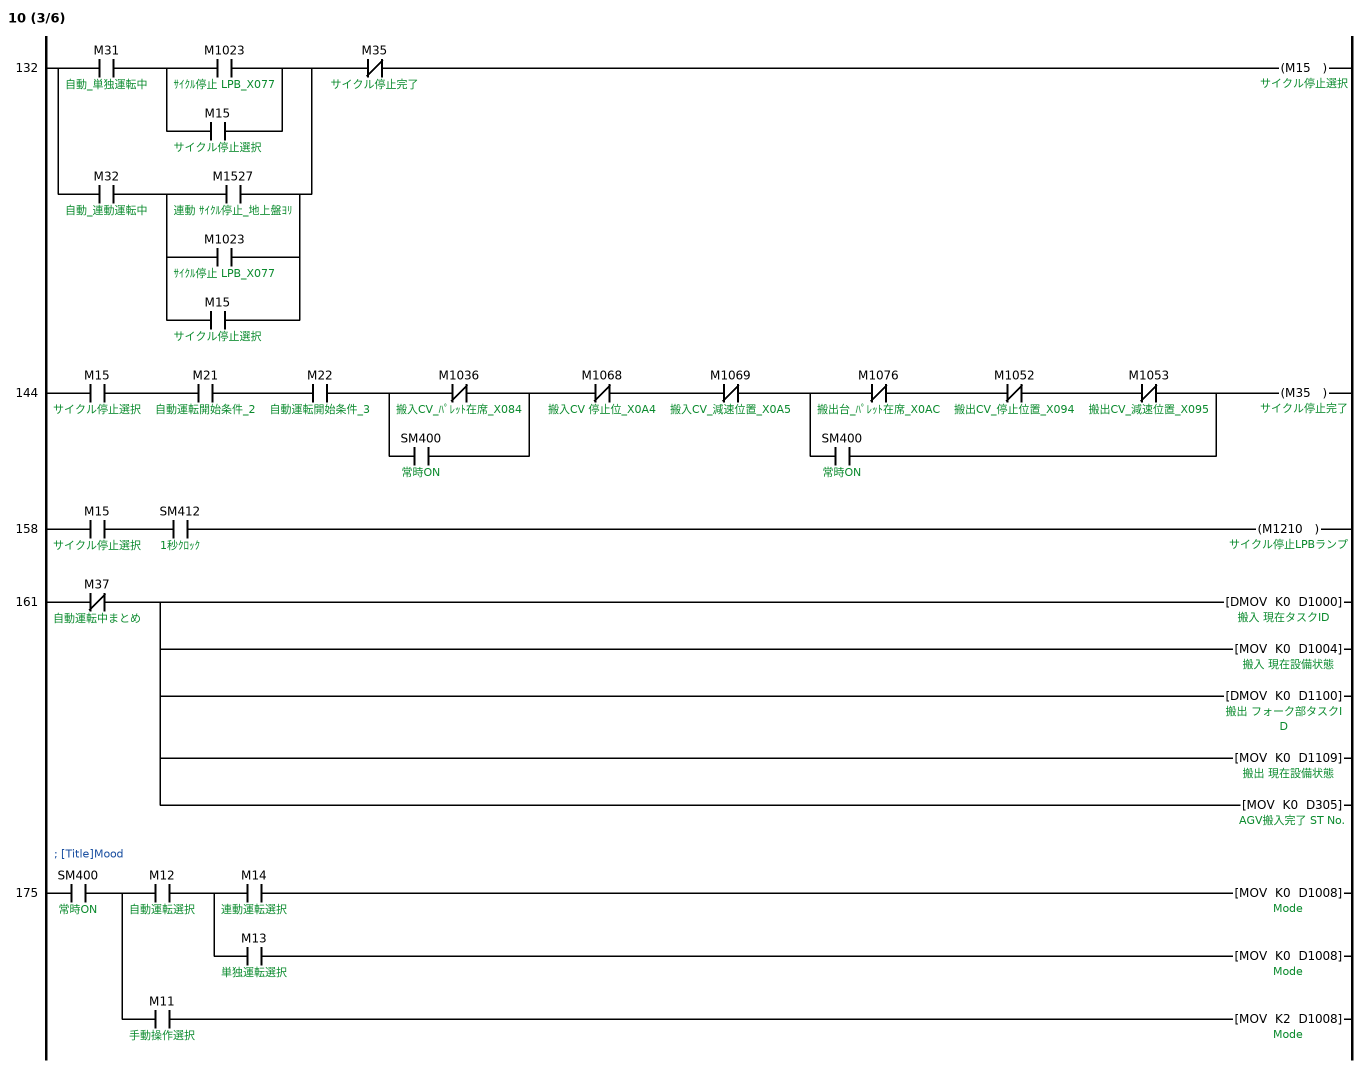
132   LD      M31  ; 自動_単独運転中
      LD      M1023  ; ｻｲｸﾙ停止 LPB_X077
      OR      M15  ; サイクル停止選択
      ANB
      LD      M32  ; 自動_連動運転中
      LD      M1527  ; 連動 ｻｲｸﾙ停止_地上盤ﾖﾘ
      OR      M1023  ; ｻｲｸﾙ停止 LPB_X077
      OR      M15  ; サイクル停止選択
      ANB
      ORB
      ANI     M35  ; サイクル停止完了
      OUT     M15  ; サイクル停止選択
144   LD      M15  ; サイクル停止選択
      AND     M21  ; 自動運転開始条件_2
      AND     M22  ; 自動運転開始条件_3
      LDI     M1036  ; 搬入CV_ﾊﾟﾚｯﾄ在席_X084
      OR      SM400  ; 常時ON
      ANB
      ANI     M1068  ; 搬入CV 停止位_X0A4
      ANI     M1069  ; 搬入CV_減速位置_X0A5
      LDI     M1076  ; 搬出台_ﾊﾟﾚｯﾄ在席_X0AC
      ANI     M1052  ; 搬出CV_停止位置_X094
      ANI     M1053  ; 搬出CV_減速位置_X095
      OR      SM400  ; 常時ON
      ANB
      OUT     M35  ; サイクル停止完了
158   LD      M15  ; サイクル停止選択
      AND     SM412  ; 1秒ｸﾛｯｸ
      OUT     M1210  ; サイクル停止LPBランプ
161   LDI     M37  ; 自動運転中まとめ
      DMOV    K0 D1000  ; 搬入 現在タスクID
      MOV     K0 D1004  ; 搬入 現在設備状態
      DMOV    K0 D1100  ; 搬出 フォーク部タスクID
      MOV     K0 D1109  ; 搬出 現在設備状態
      MOV     K0 D305  ; AGV搬入完了 ST No.
; [Title]Mood
175   LD      SM400  ; 常時ON
      MPS
      AND     M12  ; 自動運転選択
      MPS
      AND     M14  ; 連動運転選択
      MOV     K0 D1008  ; Mode
      MPP
      AND     M13  ; 単独運転選択
      MOV     K0 D1008
      MPP
      AND     M11  ; 手動操作選択
      MOV     K2 D1008
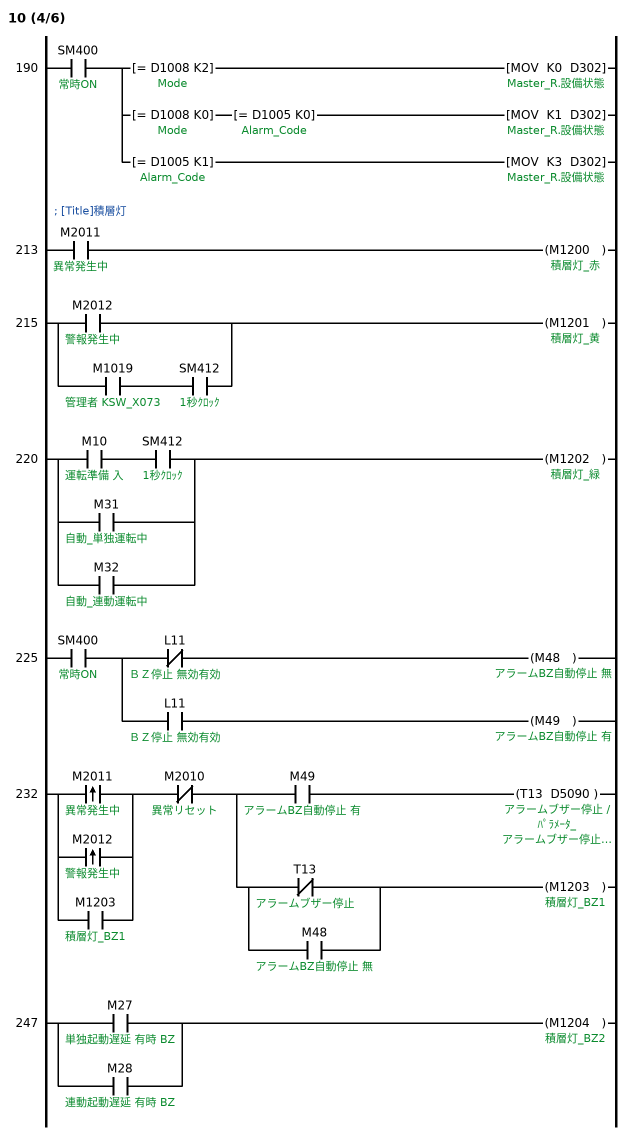
190   LD      SM400  ; 常時ON
      MPS
      AND=    D1008 K2  ; Mode
      MOV     K0 D302  ; Master_R.設備状態
      MRD
      AND=    D1008 K0  ; Mode
      AND=    D1005 K0  ; Alarm_Code
      MOV     K1 D302
      MPP
      AND=    D1005 K1  ; Alarm_Code
      MOV     K3 D302
; [Title]積層灯
213   LD      M2011  ; 異常発生中
      OUT     M1200  ; 積層灯_赤
215   LD      M2012  ; 警報発生中
      LD      M1019  ; 管理者 KSW_X073
      AND     SM412  ; 1秒ｸﾛｯｸ
      ORB
      OUT     M1201  ; 積層灯_黄
220   LD      M10  ; 運転準備 入
      AND     SM412  ; 1秒ｸﾛｯｸ
      OR      M31  ; 自動_単独運転中
      OR      M32  ; 自動_連動運転中
      OUT     M1202  ; 積層灯_緑
225   LD      SM400  ; 常時ON
      MPS
      ANI     L11  ; ＢＺ停止 無効有効
      OUT     M48  ; アラームBZ自動停止 無
      MPP
      AND     L11  ; ＢＺ停止 無効有効
      OUT     M49  ; アラームBZ自動停止 有
232   LDP     M2011  ; 異常発生中
      ORP     M2012  ; 警報発生中
      OR      M1203  ; 積層灯_BZ1
      ANI     M2010  ; 異常リセット
      MPS
      AND     M49  ; アラームBZ自動停止 有
      OUT     T13 D5090  ; アラームブザー停止 / ﾊﾟﾗﾒｰﾀ_アラームブザー停止設定値
      MPP
      LDI     T13  ; アラームブザー停止
      OR      M48  ; アラームBZ自動停止 無
      ANB
      OUT     M1203  ; 積層灯_BZ1
247   LD      M27  ; 単独起動遅延 有時 BZ
      OR      M28  ; 連動起動遅延 有時 BZ
      OUT     M1204  ; 積層灯_BZ2
